KUKA KRL program: MyProgram_298().src

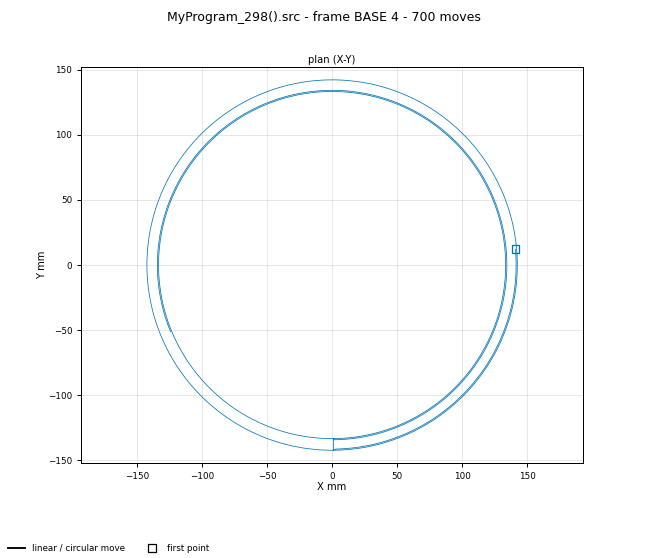
[picture p0: tool path of MyProgram_298().src in frame BASE 4, 700 of 700 moves have a stored position in this frame; points joined in program order, loops and branches not executed]
&ACCESS RVP
&REL 1
&PARAM TEMPLATE = C:\KRC\Roboter\Template\vorgabe
&PARAM EDITMASK = *
DEF MyProgram_298()
; ---- Setting reference (Base) ----
$BASE = BASE_DATA[4]

; --------------------------
; ---- Setting tool (TCP) ----
$TOOL = TOOL_DATA[3]
; --------------------------

$VEL.CP = VEL_APROX_PRINT
Startdeposition()
$VEL.CP = VEL_PRINT
LIN {X 140.7896,Y 12.0688,Z 178,A 6.9353,B 5.8277,C 0.252,E1 5.9925,E2 445.646} C_DIS
LIN {X 141.111,Y 7.4247,Z 178,A 5.2439,B 5.8277,C 0.2542,E1 5.9928,E2 447.3133} C_DIS
LIN {X 141.2495,Y 3.9929,Z 178,A 3.8231,B 5.8274,C 0.2586,E1 5.9929,E2 448.7388} C_DIS
LIN {X 141.3032,Y 0.9542,Z 178,A 2.4803,B 5.8272,C 0.2639,E1 5.9929,E2 450.0971} C_DIS
LIN {X 141.2517,Y -3.912,Z 178,A 0.8337,B 5.8272,C 0.2642,E1 5.9929,E2 451.7025} C_DIS
LIN {X 141.1557,Y -6.5363,Z 178,A -0.2484,B 5.827,C 0.2675,E1 5.9928,E2 452.7877} C_DIS
LIN {X 140.9501,Y -10.0235,Z 178,A -1.7448,B 5.8268,C 0.2729,E1 5.9925,E2 454.2957} C_DIS
LIN {X 140.6912,Y -13.1685,Z 178,A -2.8653,B 5.8268,C 0.2739,E1 5.9922,E2 455.3963} C_DIS
LIN {X 140.4174,Y -15.8362,Z 178,A -4.0893,B 5.8265,C 0.2793,E1 5.9919,E2 456.6392} C_DIS
LIN {X 139.8782,Y -20.0345,Z 178,A -5.6337,B 5.8264,C 0.2813,E1 5.9913,E2 458.1625} C_DIS
LIN {X 139.4162,Y -23.0315,Z 178,A -6.8756,B 5.8262,C 0.285,E1 5.9907,E2 459.407} C_DIS
LIN {X 138.9631,Y -25.6338,Z 178,A -7.9325,B 5.8261,C 0.2878,E1 5.9902,E2 460.4631} C_DIS
LIN {X 138.2972,Y -29.0141,Z 178,A -9.3188,B 5.8259,C 0.2915,E1 5.9895,E2 461.8492} C_DIS
LIN {X 137.5734,Y -32.2709,Z 178,A -10.7608,B 5.8256,C 0.2968,E1 5.9885,E2 463.3041} C_DIS
LIN {X 136.5863,Y -36.2143,Z 178,A -12.0709,B 5.8256,C 0.2958,E1 5.9877,E2 464.571} C_DIS
LIN {X 134.7,Y -42.6994,Z 178,A -14.9784,B 5.8251,C 0.3062,E1 5.9854,E2 467.5033} C_DIS
LIN {X 133.7418,Y -45.6164,Z 178,A -16.2242,B 5.825,C 0.3096,E1 5.9842,E2 468.7504} C_DIS
LIN {X 132.4239,Y -49.3072,Z 178,A -17.5833,B 5.825,C 0.3101,E1 5.983,E2 470.0805} C_DIS
LIN {X 131.439,Y -51.8799,Z 178,A -18.785,B 5.8247,C 0.3145,E1 5.9817,E2 471.2945} C_DIS
LIN {X 130.3827,Y -54.4752,Z 178,A -19.833,B 5.8247,C 0.3161,E1 5.9806,E2 472.3318} C_DIS
LIN {X 129.269,Y -57.0718,Z 178,A -21.1045,B 5.8243,C 0.3212,E1 5.9792,E2 473.621} C_DIS
LIN {X 127.8364,Y -60.2132,Z 178,A -22.518,B 5.8241,C 0.3251,E1 5.9775,E2 475.0377} C_DIS
LIN {X 126.2018,Y -63.5662,Z 178,A -23.9585,B 5.824,C 0.3278,E1 5.9758,E2 476.47} C_DIS
LIN {X 124.2714,Y -67.2649,Z 178,A -25.6148,B 5.8237,C 0.3316,E1 5.9736,E2 478.1232} C_DIS
LIN {X 122.0886,Y -71.1498,Z 178,A -27.2593,B 5.8237,C 0.3335,E1 5.9713,E2 479.7478} C_DIS
LIN {X 119.3608,Y -75.636,Z 178,A -29.4838,B 5.8232,C 0.3403,E1 5.9681,E2 481.987} C_DIS
LIN {X 116.8514,Y -79.4582,Z 178,A -31.2611,B 5.8231,C 0.3436,E1 5.9653,E2 483.7558} C_DIS
LIN {X 114.4302,Y -82.9065,Z 178,A -33.3278,B 5.8225,C 0.3534,E1 5.9619,E2 485.8715} C_DIS
LIN {X 111.8215,Y -86.3927,Z 178,A -34.7631,B 5.8225,C 0.3522,E1 5.9595,E2 487.2647} C_DIS
LIN {X 108.8999,Y -90.0476,Z 178,A -36.5124,B 5.8225,C 0.3542,E1 5.9564,E2 488.996} C_DIS
LIN {X 106.2988,Y -93.1042,Z 178,A -38.1229,B 5.8222,C 0.3575,E1 5.9535,E2 490.6058} C_DIS
LIN {X 103.2393,Y -96.4855,Z 178,A -39.9595,B 5.822,C 0.3613,E1 5.95,E2 492.4424} C_DIS
LIN {X 99.9844,Y -99.855,Z 178,A -41.8636,B 5.8217,C 0.3654,E1 5.9463,E2 494.3488} C_DIS
LIN {X 96.8119,Y -102.9333,Z 178,A -43.5703,B 5.8216,C 0.3677,E1 5.9429,E2 496.0457} C_DIS
LIN {X 93.3892,Y -106.0485,Z 178,A -45.543,B 5.8213,C 0.3729,E1 5.9387,E2 498.0328} C_DIS
LIN {X 89.623,Y -109.2499,Z 178,A -47.3778,B 5.8212,C 0.3741,E1 5.9349,E2 499.8468} C_DIS
LIN {X 86.4476,Y -111.7792,Z 178,A -48.9811,B 5.821,C 0.3765,E1 5.9313,E2 501.4458} C_DIS
LIN {X 82.9595,Y -114.3918,Z 178,A -50.6703,B 5.8209,C 0.3785,E1 5.9276,E2 503.1261} C_DIS
LIN {X 79.2176,Y -117.0142,Z 178,A -52.5363,B 5.8207,C 0.3818,E1 5.9233,E2 504.9954} C_DIS
LIN {X 75.9408,Y -119.1673,Z 178,A -54.1352,B 5.8205,C 0.3846,E1 5.9195,E2 506.5969} C_DIS
LIN {X 72.1514,Y -121.4989,Z 178,A -55.6674,B 5.8205,C 0.3833,E1 5.916,E2 508.0941} C_DIS
LIN {X 67.5081,Y -124.1388,Z 178,A -58.0661,B 5.8201,C 0.3901,E1 5.91,E2 510.5258} C_DIS
LIN {X 64.3589,Y -125.7982,Z 178,A -59.4105,B 5.8201,C 0.3906,E1 5.9067,E2 511.858} C_DIS
LIN {X 61.486,Y -127.2284,Z 178,A -60.7675,B 5.8199,C 0.3932,E1 5.9033,E2 513.2236} C_DIS
LIN {X 58.1815,Y -128.7726,Z 178,A -62.134,B 5.8199,C 0.3935,E1 5.8999,E2 514.5761} C_DIS
LIN {X 55.3271,Y -130.0261,Z 178,A -63.5794,B 5.8196,C 0.3977,E1 5.8961,E2 516.0468} C_DIS
LIN {X 51.3253,Y -131.6546,Z 178,A -65.0411,B 5.8198,C 0.3955,E1 5.8924,E2 517.4709} C_DIS
LIN {X 48.6469,Y -132.6698,Z 178,A -66.427,B 5.8195,C 0.4001,E1 5.8887,E2 518.8878} C_DIS
LIN {X 44.7714,Y -134.0252,Z 178,A -67.947,B 5.8195,C 0.3997,E1 5.8847,E2 520.3894} C_DIS
LIN {X 41.9416,Y -134.9389,Z 178,A -69.4697,B 5.8191,C 0.4055,E1 5.8806,E2 521.9554} C_DIS
LIN {X 38.5301,Y -135.9519,Z 178,A -70.6263,B 5.8193,C 0.4026,E1 5.8775,E2 523.0747} C_DIS
LIN {X 35.2419,Y -136.8412,Z 178,A -72.4658,B 5.8187,C 0.4104,E1 5.8724,E2 524.9762} C_DIS
LIN {X 30.6075,Y -137.9532,Z 178,A -74.0137,B 5.819,C 0.4063,E1 5.8683,E2 526.4742} C_DIS
LIN {X 27.1022,Y -138.6834,Z 178,A -75.2034,B 5.8192,C 0.4036,E1 5.8652,E2 527.6297} C_DIS
LIN {X 23.5539,Y -139.3291,Z 178,A -76.6385,B 5.8192,C 0.4041,E1 5.8612,E2 529.062} C_DIS
LIN {X 20.7157,Y -139.7809,Z 178,A -78.0954,B 5.8188,C 0.4089,E1 5.8571,E2 530.5587} C_DIS
LIN {X 16.6458,Y -140.3219,Z 178,A -79.5217,B 5.819,C 0.4063,E1 5.8532,E2 531.954} C_DIS
LIN {X 13.9017,Y -140.6208,Z 178,A -80.6337,B 5.819,C 0.4067,E1 5.8501,E2 533.0656} C_DIS
LIN {X 10.5102,Y -140.9146,Z 178,A -81.843,B 5.8191,C 0.4048,E1 5.8468,E2 534.2527} C_DIS
LIN {X 7.3431,Y -141.1151,Z 178,A -83.4444,B 5.8188,C 0.4095,E1 5.8422,E2 535.897} C_DIS
LIN {X 2.7408,Y -141.2798,Z 178,A -85.1904,B 5.8188,C 0.4082,E1 5.8374,E2 537.6277} C_DIS
LIN {X 2.7408,Y -141.2798,Z 178,A -85.1904,B 5.8188,C 0.4082,E1 5.8374,E2 537.6277} C_DIS
Enddeposition()
LIN {X 1.0318,Y -142.2048,Z 178,A -85.5763,B 5.819,C 0.4074,E1 5.8364,E2 538.0052} C_DIS
Startdeposition()
$VEL.CP = VEL_PRINT
LIN {X 3.8018,Y -142.1593,Z 178,A -84.2114,B 5.8193,C 0.4038,E1 5.8403,E2 536.606} C_DIS
LIN {X 7.0997,Y -142.0327,Z 178,A -82.8414,B 5.8193,C 0.4029,E1 5.8442,E2 535.2298} C_DIS
LIN {X 10.5794,Y -141.8161,Z 178,A -81.4286,B 5.8193,C 0.4023,E1 5.8481,E2 533.8152} C_DIS
LIN {X 13.9421,Y -141.5253,Z 178,A -80.075,B 5.8194,C 0.4019,E1 5.8519,E2 532.4617} C_DIS
LIN {X 17.7286,Y -141.1026,Z 178,A -78.5776,B 5.8194,C 0.4017,E1 5.856,E2 530.9687} C_DIS
LIN {X 20.9908,Y -140.6543,Z 178,A -77.2417,B 5.8194,C 0.4009,E1 5.8597,E2 529.6307} C_DIS
LIN {X 24.3237,Y -140.1162,Z 178,A -75.8217,B 5.8196,C 0.3992,E1 5.8636,E2 528.2017} C_DIS
LIN {X 27.858,Y -139.4554,Z 178,A -74.418,B 5.8196,C 0.3989,E1 5.8675,E2 526.8033} C_DIS
LIN {X 31.2944,Y -138.7243,Z 178,A -73.0141,B 5.8196,C 0.398,E1 5.8713,E2 525.4001} C_DIS
LIN {X 34.5683,Y -137.945,Z 178,A -71.6294,B 5.8198,C 0.3965,E1 5.8751,E2 524.0105} C_DIS
LIN {X 37.9249,Y -137.0601,Z 178,A -70.2819,B 5.8198,C 0.3961,E1 5.8787,E2 522.6691} C_DIS
LIN {X 41.789,Y -135.9313,Z 178,A -68.5849,B 5.82,C 0.3934,E1 5.8833,E2 520.9607} C_DIS
LIN {X 46.3797,Y -134.4342,Z 178,A -66.7442,B 5.82,C 0.393,E1 5.8881,E2 519.133} C_DIS
LIN {X 49.5577,Y -133.2956,Z 178,A -65.3978,B 5.82,C 0.3918,E1 5.8916,E2 517.7874} C_DIS
LIN {X 52.8099,Y -132.041,Z 178,A -64.0082,B 5.8202,C 0.3904,E1 5.8953,E2 516.3989} C_DIS
LIN {X 56.0719,Y -130.6892,Z 178,A -62.5985,B 5.8202,C 0.3888,E1 5.8989,E2 514.9898} C_DIS
LIN {X 59.2173,Y -129.2947,Z 178,A -61.2162,B 5.8204,C 0.3871,E1 5.9024,E2 513.607} C_DIS
LIN {X 62.3694,Y -127.8044,Z 178,A -59.845,B 5.8204,C 0.3857,E1 5.9058,E2 512.2393} C_DIS
LIN {X 65.496,Y -126.2311,Z 178,A -58.3602,B 5.8207,C 0.3826,E1 5.9096,E2 510.7433} C_DIS
LIN {X 69.4042,Y -124.1261,Z 178,A -56.6109,B 5.8208,C 0.3806,E1 5.9138,E2 508.998} C_DIS
LIN {X 73.1252,Y -121.9711,Z 178,A -54.9593,B 5.8209,C 0.3792,E1 5.9178,E2 507.356} C_DIS
LIN {X 76.0902,Y -120.1435,Z 178,A -53.5759,B 5.821,C 0.3772,E1 5.9211,E2 505.9741} C_DIS
LIN {X 79.0543,Y -118.214,Z 178,A -52.0494,B 5.8213,C 0.3732,E1 5.9246,E2 504.4326} C_DIS
LIN {X 82.6534,Y -115.7261,Z 178,A -50.4466,B 5.8213,C 0.3727,E1 5.9283,E2 502.8502} C_DIS
LIN {X 85.4653,Y -113.6656,Z 178,A -49.0809,B 5.8215,C 0.3708,E1 5.9313,E2 501.4885} C_DIS
LIN {X 88.6759,Y -111.1788,Z 178,A -47.4079,B 5.8217,C 0.3672,E1 5.935,E2 499.809} C_DIS
LIN {X 92.181,Y -108.2903,Z 178,A -45.6378,B 5.8218,C 0.3647,E1 5.9388,E2 498.0455} C_DIS
LIN {X 94.862,Y -105.9496,Z 178,A -44.2317,B 5.822,C 0.3623,E1 5.9417,E2 496.642} C_DIS
LIN {X 97.4308,Y -103.5925,Z 178,A -42.8526,B 5.8221,C 0.3598,E1 5.9445,E2 495.265} C_DIS
LIN {X 100.5199,Y -100.5984,Z 178,A -41.1447,B 5.8223,C 0.3567,E1 5.9479,E2 493.5591} C_DIS
LIN {X 103.0441,Y -98.0109,Z 178,A -39.729,B 5.8225,C 0.3542,E1 5.9507,E2 492.1476} C_DIS
LIN {X 105.4161,Y -95.4546,Z 178,A -38.3467,B 5.8227,C 0.3515,E1 5.9533,E2 490.7671} C_DIS
LIN {X 108.2186,Y -92.2654,Z 178,A -36.6624,B 5.8229,C 0.3482,E1 5.9564,E2 489.0848} C_DIS
LIN {X 110.5175,Y -89.499,Z 178,A -35.2473,B 5.823,C 0.3454,E1 5.9589,E2 487.673} C_DIS
LIN {X 112.6968,Y -86.7395,Z 178,A -33.7189,B 5.8233,C 0.3403,E1 5.9615,E2 486.1283} C_DIS
LIN {X 115.2677,Y -83.2918,Z 178,A -32.1596,B 5.8233,C 0.3391,E1 5.964,E2 484.5909} C_DIS
LIN {X 117.568,Y -80.0126,Z 178,A -30.4755,B 5.8237,C 0.3341,E1 5.9667,E2 482.8958} C_DIS
LIN {X 120.1428,Y -76.0912,Z 178,A -28.722,B 5.8238,C 0.3317,E1 5.9694,E2 481.159} C_DIS
LIN {X 122.116,Y -72.8822,Z 178,A -27.153,B 5.8241,C 0.327,E1 5.9716,E2 479.5816} C_DIS
LIN {X 124.1647,Y -69.3355,Z 178,A -25.5171,B 5.8243,C 0.3231,E1 5.9739,E2 477.9462} C_DIS
LIN {X 126.2634,Y -65.4346,Z 178,A -23.8758,B 5.8244,C 0.3209,E1 5.976,E2 476.3226} C_DIS
LIN {X 127.8295,Y -62.3186,Z 178,A -22.5037,B 5.8246,C 0.3178,E1 5.9777,E2 474.9537} C_DIS
LIN {X 129.3183,Y -59.1663,Z 178,A -21.1285,B 5.8248,C 0.3146,E1 5.9793,E2 473.5811} C_DIS
LIN {X 130.7514,Y -55.9279,Z 178,A -19.7382,B 5.8249,C 0.3114,E1 5.9809,E2 472.1945} C_DIS
LIN {X 132.0827,Y -52.7065,Z 178,A -18.3668,B 5.8251,C 0.3082,E1 5.9823,E2 470.8262} C_DIS
LIN {X 133.2951,Y -49.559,Z 178,A -17.0401,B 5.8253,C 0.3051,E1 5.9836,E2 469.5027} C_DIS
LIN {X 134.5104,Y -46.1599,Z 178,A -15.4987,B 5.8255,C 0.2997,E1 5.985,E2 467.9482} C_DIS
LIN {X 135.5815,Y -42.9116,Z 178,A -14.2649,B 5.8256,C 0.2983,E1 5.9861,E2 466.7327} C_DIS
LIN {X 136.6219,Y -39.4755,Z 178,A -12.8713,B 5.8258,C 0.2952,E1 5.9872,E2 465.3449} C_DIS
LIN {X 137.5474,Y -36.1194,Z 178,A -11.5022,B 5.8259,C 0.2919,E1 5.9882,E2 463.9791} C_DIS
LIN {X 138.3645,Y -32.8501,Z 178,A -10.1385,B 5.8261,C 0.288,E1 5.9891,E2 462.6133} C_DIS
LIN {X 139.1267,Y -29.4571,Z 178,A -8.8032,B 5.8263,C 0.2851,E1 5.9898,E2 461.2857} C_DIS
LIN {X 139.8334,Y -25.9021,Z 178,A -7.3729,B 5.8264,C 0.2815,E1 5.9906,E2 459.8581} C_DIS
LIN {X 140.4073,Y -22.5855,Z 178,A -6.0384,B 5.8266,C 0.2781,E1 5.9912,E2 458.5254} C_DIS
LIN {X 140.9181,Y -19.1361,Z 178,A -4.6369,B 5.8268,C 0.2741,E1 5.9918,E2 457.1232} C_DIS
LIN {X 141.356,Y -15.5658,Z 178,A -3.283,B 5.8269,C 0.2716,E1 5.9922,E2 455.7808} C_DIS
LIN {X 141.7303,Y -11.675,Z 178,A -1.7851,B 5.8271,C 0.2684,E1 5.9926,E2 454.2919} C_DIS
LIN {X 141.943,Y -8.7115,Z 178,A -0.5464,B 5.8272,C 0.2643,E1 5.9928,E2 453.0466} C_DIS
LIN {X 142.1185,Y -5.1195,Z 178,A 0.8518,B 5.8274,C 0.261,E1 5.993,E2 451.654} C_DIS
LIN {X 142.2072,Y -0.9928,Z 178,A 2.268,B 5.8274,C 0.2604,E1 5.993,E2 450.2694} C_DIS
LIN {X 142.199,Y 1.8524,Z 178,A 3.5882,B 5.8277,C 0.2542,E1 5.993,E2 448.9252} C_DIS
LIN {X 142.1137,Y 5.2435,Z 178,A 4.9594,B 5.8279,C 0.2502,E1 5.9929,E2 447.5523} C_DIS
LIN {X 141.8893,Y 9.577,Z 178,A 6.8418,B 5.8282,C 0.243,E1 5.9926,E2 445.6507} C_DIS
LIN {X 141.5259,Y 13.9363,Z 178,A 8.3626,B 5.8282,C 0.242,E1 5.9922,E2 444.1608} C_DIS
LIN {X 141.1269,Y 17.531,Z 178,A 9.7666,B 5.8283,C 0.2388,E1 5.9917,E2 442.7628} C_DIS
LIN {X 140.6554,Y 20.984,Z 178,A 11.1263,B 5.8285,C 0.2355,E1 5.9912,E2 441.4081} C_DIS
LIN {X 140.1177,Y 24.3154,Z 178,A 12.5193,B 5.8286,C 0.2312,E1 5.9905,E2 440.0097} C_DIS
LIN {X 139.4419,Y 27.9246,Z 178,A 13.9069,B 5.8288,C 0.2285,E1 5.9898,E2 438.6332} C_DIS
LIN {X 138.7328,Y 31.2573,Z 178,A 15.2662,B 5.8288,C 0.2249,E1 5.989,E2 437.2747} C_DIS
LIN {X 137.9528,Y 34.5376,Z 178,A 16.62,B 5.829,C 0.2213,E1 5.9881,E2 435.9207} C_DIS
LIN {X 136.8515,Y 38.6708,Z 178,A 18.1868,B 5.8291,C 0.2191,E1 5.987,E2 434.3735} C_DIS
LIN {X 136.0528,Y 41.392,Z 178,A 19.3635,B 5.8293,C 0.2154,E1 5.986,E2 433.1915} C_DIS
LIN {X 135.032,Y 44.6102,Z 178,A 20.7434,B 5.8293,C 0.2114,E1 5.9848,E2 431.8083} C_DIS
LIN {X 133.8596,Y 48.013,Z 178,A 22.1484,B 5.8295,C 0.2083,E1 5.9835,E2 430.4084} C_DIS
LIN {X 132.6757,Y 51.1942,Z 178,A 23.47,B 5.8296,C 0.2054,E1 5.9822,E2 429.0921} C_DIS
LIN {X 131.3819,Y 54.4291,Z 178,A 24.8413,B 5.8297,C 0.2022,E1 5.9808,E2 427.7242} C_DIS
LIN {X 129.9867,Y 57.6818,Z 178,A 26.3148,B 5.8299,C 0.1977,E1 5.9791,E2 426.2437} C_DIS
LIN {X 128.5349,Y 60.8488,Z 178,A 27.5899,B 5.8299,C 0.1962,E1 5.9776,E2 424.9848} C_DIS
LIN {X 127.0309,Y 63.9307,Z 178,A 28.9598,B 5.83,C 0.1928,E1 5.9759,E2 423.6159} C_DIS
LIN {X 125.3934,Y 67.0872,Z 178,A 30.4698,B 5.8302,C 0.188,E1 5.9739,E2 422.095} C_DIS
LIN {X 123.3001,Y 70.8619,Z 178,A 32.0718,B 5.8302,C 0.1859,E1 5.9718,E2 420.5102} C_DIS
LIN {X 121.5257,Y 73.863,Z 178,A 33.4534,B 5.8304,C 0.1828,E1 5.9698,E2 419.131} C_DIS
LIN {X 119.2361,Y 77.504,Z 178,A 35.159,B 5.8304,C 0.1791,E1 5.9672,E2 417.4282} C_DIS
LIN {X 116.8061,Y 81.1201,Z 178,A 36.8825,B 5.8306,C 0.1754,E1 5.9645,E2 415.7083} C_DIS
LIN {X 114.7097,Y 84.0585,Z 178,A 38.3768,B 5.8307,C 0.1714,E1 5.9621,E2 414.2082} C_DIS
LIN {X 112.0833,Y 87.5306,Z 178,A 40.0033,B 5.8307,C 0.1695,E1 5.9593,E2 412.5978} C_DIS
LIN {X 109.8763,Y 90.2855,Z 178,A 41.5412,B 5.8309,C 0.1645,E1 5.9566,E2 411.0444} C_DIS
LIN {X 107.042,Y 93.6278,Z 178,A 43.2608,B 5.8309,C 0.1614,E1 5.9534,E2 409.3302} C_DIS
LIN {X 104.1886,Y 96.793,Z 178,A 44.8289,B 5.831,C 0.1601,E1 5.9505,E2 407.7811} C_DIS
LIN {X 101.7452,Y 99.3586,Z 178,A 46.2987,B 5.8311,C 0.1565,E1 5.9477,E2 406.3055} C_DIS
LIN {X 98.6592,Y 102.4237,Z 178,A 47.9572,B 5.8311,C 0.1545,E1 5.9444,E2 404.6588} C_DIS
LIN {X 95.5257,Y 105.3516,Z 178,A 49.6621,B 5.8313,C 0.1514,E1 5.9409,E2 402.9565} C_DIS
LIN {X 91.9966,Y 108.4471,Z 178,A 51.602,B 5.8313,C 0.1472,E1 5.9368,E2 401.01} C_DIS
LIN {X 88.8163,Y 111.067,Z 178,A 53.1334,B 5.8313,C 0.1461,E1 5.9335,E2 399.4951} C_DIS
LIN {X 86.1098,Y 113.1784,Z 178,A 54.5078,B 5.8314,C 0.1438,E1 5.9304,E2 398.1216} C_DIS
LIN {X 83.3077,Y 115.2561,Z 178,A 56.015,B 5.8315,C 0.1399,E1 5.927,E2 396.6011} C_DIS
LIN {X 79.7275,Y 117.761,Z 178,A 57.622,B 5.8315,C 0.1393,E1 5.9234,E2 395.0139} C_DIS
LIN {X 76.7708,Y 119.7096,Z 178,A 59.0155,B 5.8315,C 0.1376,E1 5.9201,E2 393.6246} C_DIS
LIN {X 73.8139,Y 121.5554,Z 178,A 60.4867,B 5.8317,C 0.1345,E1 5.9166,E2 392.1448} C_DIS
LIN {X 70.0937,Y 123.7384,Z 178,A 62.2577,B 5.8317,C 0.1315,E1 5.9123,E2 390.3695} C_DIS
LIN {X 66.2699,Y 125.8248,Z 178,A 63.8719,B 5.8317,C 0.1311,E1 5.9084,E2 388.7734} C_DIS
LIN {X 63.0883,Y 127.4498,Z 178,A 65.2721,B 5.8317,C 0.1298,E1 5.9049,E2 387.3783} C_DIS
LIN {X 59.9571,Y 128.9527,Z 178,A 66.6575,B 5.8318,C 0.1283,E1 5.9014,E2 385.9949} C_DIS
LIN {X 57.5272,Y 130.0558,Z 178,A 67.7427,B 5.8318,C 0.1269,E1 5.8986,E2 384.9085} C_DIS
LIN {X 53.9852,Y 131.5672,Z 178,A 69.2765,B 5.8318,C 0.1254,E1 5.8947,E2 383.3772} C_DIS
LIN {X 51.072,Y 132.7233,Z 178,A 70.5185,B 5.8318,C 0.1243,E1 5.8914,E2 382.138} C_DIS
LIN {X 47.2351,Y 134.1376,Z 178,A 72.2781,B 5.832,C 0.1211,E1 5.8868,E2 380.3642} C_DIS
LIN {X 43.3592,Y 135.4385,Z 178,A 73.8744,B 5.832,C 0.1203,E1 5.8826,E2 378.7748} C_DIS
LIN {X 39.5047,Y 136.6133,Z 178,A 75.4664,B 5.832,C 0.1194,E1 5.8783,E2 377.1871} C_DIS
LIN {X 36.119,Y 137.5475,Z 178,A 76.8008,B 5.832,C 0.1194,E1 5.8747,E2 375.8635} C_DIS
LIN {X 32.8433,Y 138.3661,Z 178,A 78.159,B 5.832,C 0.1185,E1 5.871,E2 374.5059} C_DIS
LIN {X 29.4441,Y 139.1295,Z 178,A 79.5529,B 5.832,C 0.1178,E1 5.8672,E2 373.1137} C_DIS
LIN {X 25.9185,Y 139.8303,Z 178,A 80.9981,B 5.832,C 0.117,E1 5.8633,E2 371.6693} C_DIS
LIN {X 22.2652,Y 140.457,Z 178,A 82.3946,B 5.832,C 0.1176,E1 5.8595,E2 370.2857} C_DIS
LIN {X 19.1288,Y 140.9191,Z 178,A 83.8019,B 5.832,C 0.1153,E1 5.8555,E2 368.8621} C_DIS
LIN {X 15.557,Y 141.3569,Z 178,A 85.1854,B 5.832,C 0.1156,E1 5.8517,E2 367.4876} C_DIS
LIN {X 12.1982,Y 141.6861,Z 178,A 86.5867,B 5.832,C 0.1147,E1 5.8478,E2 366.0814} C_DIS
LIN {X 8.7224,Y 141.9423,Z 178,A 87.9783,B 5.832,C 0.1145,E1 5.8439,E2 364.692} C_DIS
LIN {X 5.1123,Y 142.1188,Z 178,A 89.3938,B 5.832,C 0.1149,E1 5.84,E2 363.2824} C_DIS
LIN {X 1.6282,Y 142.2027,Z 178,A 90.795,B 5.832,C 0.1148,E1 5.8361,E2 361.8822} C_DIS
LIN {X -1.8595,Y 142.1989,Z 178,A 92.2118,B 5.832,C 0.1146,E1 5.8321,E2 360.4646} C_DIS
LIN {X -5.2331,Y 142.1141,Z 178,A 93.6179,B 5.8321,C 0.1141,E1 5.8282,E2 359.053} C_DIS
LIN {X -8.7251,Y 141.9421,Z 178,A 95.014,B 5.8321,C 0.1144,E1 5.8243,E2 357.6592} C_DIS
LIN {X -12.3225,Y 141.6756,Z 178,A 96.4505,B 5.8321,C 0.1149,E1 5.8203,E2 356.2256} C_DIS
LIN {X -15.6804,Y 141.3436,Z 178,A 97.812,B 5.8321,C 0.1153,E1 5.8165,E2 354.8646} C_DIS
LIN {X -19.2495,Y 140.9032,Z 178,A 99.2796,B 5.8321,C 0.1155,E1 5.8125,E2 353.3954} C_DIS
LIN {X -22.6275,Y 140.4004,Z 178,A 100.6613,B 5.8321,C 0.116,E1 5.8086,E2 352.0137} C_DIS
LIN {X -26.1702,Y 139.7821,Z 178,A 102.11,B 5.8321,C 0.1167,E1 5.8047,E2 350.5659} C_DIS
LIN {X -29.5798,Y 139.1002,Z 178,A 103.5149,B 5.8321,C 0.1174,E1 5.8008,E2 349.1613} C_DIS
LIN {X -32.9661,Y 138.3365,Z 178,A 104.8898,B 5.8321,C 0.1186,E1 5.7971,E2 347.7902} C_DIS
LIN {X -36.3319,Y 137.4907,Z 178,A 106.3064,B 5.832,C 0.1193,E1 5.7933,E2 346.3721} C_DIS
LIN {X -39.9883,Y 136.4717,Z 178,A 107.8081,B 5.832,C 0.1208,E1 5.7892,E2 344.8749} C_DIS
LIN {X -42.95,Y 135.5692,Z 178,A 109.1216,B 5.832,C 0.121,E1 5.7857,E2 343.5538} C_DIS
LIN {X -46.3741,Y 134.4361,Z 178,A 110.5892,B 5.832,C 0.1221,E1 5.7818,E2 342.0852} C_DIS
LIN {X -49.5676,Y 133.2919,Z 178,A 112.0314,B 5.832,C 0.1225,E1 5.778,E2 340.6343} C_DIS
LIN {X -52.8178,Y 132.0378,Z 178,A 113.3778,B 5.8319,C 0.1247,E1 5.7745,E2 339.2962} C_DIS
LIN {X -56.0356,Y 130.7049,Z 178,A 114.8084,B 5.8319,C 0.1259,E1 5.7709,E2 337.8631} C_DIS
LIN {X -59.2195,Y 129.2937,Z 178,A 116.2254,B 5.8319,C 0.1273,E1 5.7672,E2 336.4454} C_DIS
LIN {X -62.3688,Y 127.8047,Z 178,A 117.6316,B 5.8318,C 0.129,E1 5.7637,E2 335.0398} C_DIS
LIN {X -65.4985,Y 126.2298,Z 178,A 119.0537,B 5.8318,C 0.1307,E1 5.7602,E2 333.6175} C_DIS
LIN {X -68.623,Y 124.5596,Z 178,A 120.4854,B 5.8318,C 0.1325,E1 5.7567,E2 332.1864} C_DIS
LIN {X -71.6092,Y 122.8675,Z 178,A 121.9101,B 5.8317,C 0.134,E1 5.7532,E2 330.7572} C_DIS
LIN {X -74.6483,Y 121.0449,Z 178,A 123.3484,B 5.8317,C 0.136,E1 5.7498,E2 329.3187} C_DIS
LIN {X -77.5943,Y 119.1775,Z 178,A 124.7777,B 5.8316,C 0.1378,E1 5.7464,E2 327.8874} C_DIS
LIN {X -80.629,Y 117.1457,Z 178,A 126.3956,B 5.8316,C 0.1385,E1 5.7426,E2 326.2518} C_DIS
LIN {X -84.0833,Y 114.6915,Z 178,A 127.9956,B 5.8315,C 0.1425,E1 5.739,E2 324.6671} C_DIS
LIN {X -86.8207,Y 112.634,Z 178,A 129.3938,B 5.8315,C 0.1447,E1 5.7359,E2 323.2676} C_DIS
LIN {X -89.5924,Y 110.4422,Z 178,A 130.8551,B 5.8314,C 0.1468,E1 5.7327,E2 321.8026} C_DIS
LIN {X -92.2978,Y 108.191,Z 178,A 132.4283,B 5.8314,C 0.1477,E1 5.7293,E2 320.2106} C_DIS
LIN {X -95.5623,Y 105.3184,Z 178,A 134.201,B 5.8313,C 0.1508,E1 5.7256,E2 318.4366} C_DIS
LIN {X -98.74,Y 102.3455,Z 178,A 135.9818,B 5.8312,C 0.1539,E1 5.722,E2 316.6538} C_DIS
LIN {X -101.7853,Y 99.3176,Z 178,A 137.632,B 5.8311,C 0.1583,E1 5.7188,E2 315.0155} C_DIS
LIN {X -104.2254,Y 96.7535,Z 178,A 139.0775,B 5.8311,C 0.161,E1 5.7161,E2 313.5687} C_DIS
LIN {X -106.5991,Y 94.1316,Z 178,A 140.6525,B 5.831,C 0.1624,E1 5.7131,E2 311.9755} C_DIS
LIN {X -109.3867,Y 90.8775,Z 178,A 142.2987,B 5.8308,C 0.167,E1 5.7102,E2 310.3412} C_DIS
LIN {X -111.6042,Y 88.1406,Z 178,A 143.7183,B 5.8308,C 0.1702,E1 5.7077,E2 308.9229} C_DIS
LIN {X -114.1733,Y 84.7857,Z 178,A 145.4784,B 5.8306,C 0.1735,E1 5.7047,E2 307.1568} C_DIS
LIN {X -116.2702,Y 81.8863,Z 178,A 146.9347,B 5.8306,C 0.1766,E1 5.7023,E2 305.6999} C_DIS
LIN {X -118.2437,Y 79.0098,Z 178,A 148.3807,B 5.8305,C 0.1795,E1 5.7001,E2 304.2498} C_DIS
LIN {X -120.1518,Y 76.0769,Z 178,A 149.818,B 5.8304,C 0.1826,E1 5.6979,E2 302.8103} C_DIS
LIN {X -122.0099,Y 73.0602,Z 178,A 151.2626,B 5.8303,C 0.1859,E1 5.6958,E2 301.3647} C_DIS
LIN {X -123.7376,Y 70.0951,Z 178,A 152.6857,B 5.8302,C 0.1889,E1 5.6938,E2 299.9376} C_DIS
LIN {X -125.4359,Y 67.008,Z 178,A 154.1502,B 5.8301,C 0.192,E1 5.6919,E2 298.4685} C_DIS
LIN {X -127.0653,Y 63.863,Z 178,A 155.5984,B 5.83,C 0.1955,E1 5.69,E2 297.0188} C_DIS
LIN {X -128.5902,Y 60.7331,Z 178,A 157.1545,B 5.8299,C 0.1975,E1 5.6881,E2 295.444} C_DIS
LIN {X -130.0582,Y 57.5219,Z 178,A 158.4855,B 5.8297,C 0.2021,E1 5.6866,E2 294.1262} C_DIS
LIN {X -131.4245,Y 54.327,Z 178,A 159.9187,B 5.8297,C 0.2055,E1 5.6851,E2 292.6899} C_DIS
LIN {X -132.7224,Y 51.0741,Z 178,A 161.3508,B 5.8295,C 0.209,E1 5.6836,E2 291.2563} C_DIS
LIN {X -133.8959,Y 47.9121,Z 178,A 162.7641,B 5.8294,C 0.2121,E1 5.6823,E2 289.837} C_DIS
LIN {X -135.0686,Y 44.5003,Z 178,A 164.229,B 5.8292,C 0.2159,E1 5.681,E2 288.372} C_DIS
LIN {X -136.1189,Y 41.176,Z 178,A 165.677,B 5.8292,C 0.2193,E1 5.6798,E2 286.9195} C_DIS
LIN {X -137.0573,Y 37.9346,Z 178,A 167.0802,B 5.829,C 0.2226,E1 5.6787,E2 285.5118} C_DIS
LIN {X -137.9463,Y 34.5632,Z 178,A 168.5089,B 5.8288,C 0.2263,E1 5.6777,E2 284.0812} C_DIS
LIN {X -138.8779,Y 30.6095,Z 178,A 170.0941,B 5.8286,C 0.2314,E1 5.6767,E2 282.5041} C_DIS
LIN {X -139.4861,Y 27.7076,Z 178,A 171.4085,B 5.8286,C 0.2335,E1 5.676,E2 281.1751} C_DIS
LIN {X -140.1411,Y 24.1817,Z 178,A 172.8685,B 5.8284,C 0.2374,E1 5.6753,E2 279.7144} C_DIS
LIN {X -140.6746,Y 20.8532,Z 178,A 174.2984,B 5.8283,C 0.2405,E1 5.6746,E2 278.2762} C_DIS
LIN {X -141.1546,Y 17.2988,Z 178,A 175.7859,B 5.8281,C 0.2442,E1 5.6741,E2 276.7843} C_DIS
LIN {X -141.5287,Y 13.9075,Z 178,A 177.1841,B 5.828,C 0.2478,E1 5.6737,E2 275.3841} C_DIS
LIN {X -141.8345,Y 10.328,Z 178,A 178.6416,B 5.8278,C 0.2518,E1 5.6734,E2 273.9265} C_DIS
LIN {X -142.045,Y 6.8548,Z 178,A -179.9112,B 5.8276,C 0.2554,E1 5.6732,E2 272.4745} C_DIS
LIN {X -142.168,Y 3.4889,Z 178,A -178.4178,B 5.8276,C 0.2579,E1 5.673,E2 270.9642} C_DIS
LIN {X -142.2123,Y -0.0237,Z 178,A -176.9975,B 5.8274,C 0.2618,E1 5.673,E2 269.5444} C_DIS
LIN {X -142.1674,Y -3.5132,Z 178,A -175.6025,B 5.8272,C 0.266,E1 5.6731,E2 268.152} C_DIS
LIN {X -142.0326,Y -7.102,Z 178,A -174.1506,B 5.827,C 0.27,E1 5.6733,E2 266.7005} C_DIS
LIN {X -141.8166,Y -10.5734,Z 178,A -172.691,B 5.8268,C 0.2734,E1 5.6736,E2 265.2342} C_DIS
LIN {X -141.5165,Y -14.0338,Z 178,A -171.2697,B 5.8267,C 0.2772,E1 5.6739,E2 263.811} C_DIS
LIN {X -141.1207,Y -17.5831,Z 178,A -169.7956,B 5.8265,C 0.2809,E1 5.6744,E2 262.3334} C_DIS
LIN {X -140.6498,Y -21.0198,Z 178,A -168.3818,B 5.8263,C 0.2846,E1 5.675,E2 260.9185} C_DIS
LIN {X -140.0696,Y -24.5843,Z 178,A -166.8986,B 5.8261,C 0.2884,E1 5.6757,E2 259.4325} C_DIS
LIN {X -139.456,Y -27.8551,Z 178,A -165.4784,B 5.826,C 0.2913,E1 5.6764,E2 258.0028} C_DIS
LIN {X -138.7306,Y -31.267,Z 178,A -164.0402,B 5.8258,C 0.2949,E1 5.6773,E2 256.5611} C_DIS
LIN {X -137.9493,Y -34.5516,Z 178,A -162.6164,B 5.8256,C 0.298,E1 5.6782,E2 255.1297} C_DIS
LIN {X -137.0568,Y -37.9364,Z 178,A -161.1406,B 5.8255,C 0.3012,E1 5.6793,E2 253.6461} C_DIS
LIN {X -136.053,Y -41.3912,Z 178,A -159.7478,B 5.8252,C 0.3057,E1 5.6804,E2 252.2618} C_DIS
LIN {X -135.0327,Y -44.6081,Z 178,A -158.2209,B 5.8252,C 0.3076,E1 5.6818,E2 250.7135} C_DIS
LIN {X -133.8454,Y -48.0524,Z 178,A -156.8532,B 5.8249,C 0.3126,E1 5.683,E2 249.36} C_DIS
LIN {X -132.6699,Y -51.2091,Z 178,A -155.4399,B 5.8247,C 0.3155,E1 5.6844,E2 247.94} C_DIS
LIN {X -131.3803,Y -54.4329,Z 178,A -154.0098,B 5.8245,C 0.3189,E1 5.6859,E2 246.5065} C_DIS
LIN {X -129.9904,Y -57.6735,Z 178,A -152.5673,B 5.8243,C 0.3223,E1 5.6876,E2 245.0619} C_DIS
LIN {X -128.5316,Y -60.8558,Z 178,A -151.131,B 5.8242,C 0.3256,E1 5.6893,E2 243.6229} C_DIS
LIN {X -127.0262,Y -63.9398,Z 178,A -149.7028,B 5.824,C 0.3286,E1 5.691,E2 242.1893} C_DIS
LIN {X -125.382,Y -67.1084,Z 178,A -148.229,B 5.8238,C 0.3318,E1 5.693,E2 240.7115} C_DIS
LIN {X -123.3258,Y -70.8169,Z 178,A -146.4691,B 5.8236,C 0.3354,E1 5.6954,E2 238.9454} C_DIS
LIN {X -121.5264,Y -73.8618,Z 178,A -145.0136,B 5.8234,C 0.3385,E1 5.6975,E2 237.4866} C_DIS
LIN {X -119.233,Y -77.5088,Z 178,A -143.2325,B 5.8232,C 0.3421,E1 5.7002,E2 235.7} C_DIS
LIN {X -116.8013,Y -81.1271,Z 178,A -141.4387,B 5.823,C 0.3458,E1 5.703,E2 233.902} C_DIS
LIN {X -114.7109,Y -84.0569,Z 178,A -139.9842,B 5.8228,C 0.349,E1 5.7054,E2 232.4474} C_DIS
LIN {X -112.6493,Y -86.801,Z 178,A -138.5721,B 5.8226,C 0.3517,E1 5.7078,E2 231.0319} C_DIS
LIN {X -110.4513,Y -89.5811,Z 178,A -137.1143,B 5.8225,C 0.3545,E1 5.7103,E2 229.5705} C_DIS
LIN {X -108.2098,Y -92.2756,Z 178,A -135.5352,B 5.8225,C 0.3556,E1 5.7132,E2 227.9694} C_DIS
LIN {X -105.331,Y -95.5484,Z 178,A -133.7561,B 5.8222,C 0.3589,E1 5.7165,E2 226.1876} C_DIS
LIN {X -102.223,Y -98.8665,Z 178,A -131.9257,B 5.822,C 0.3626,E1 5.72,E2 224.3579} C_DIS
LIN {X -99.3206,Y -101.7825,Z 178,A -130.3251,B 5.8217,C 0.3665,E1 5.7232,E2 222.7653} C_DIS
LIN {X -96.7954,Y -104.1864,Z 178,A -128.7959,B 5.8217,C 0.3676,E1 5.7264,E2 221.2196} C_DIS
LIN {X -93.5431,Y -107.1159,Z 178,A -127.1084,B 5.8214,C 0.3717,E1 5.7299,E2 219.5427} C_DIS
LIN {X -90.2592,Y -109.8978,Z 178,A -125.3356,B 5.8212,C 0.3743,E1 5.7337,E2 217.7649} C_DIS
LIN {X -87.3206,Y -112.2466,Z 178,A -123.7034,B 5.8212,C 0.3755,E1 5.7373,E2 216.1171} C_DIS
LIN {X -84.0043,Y -114.7495,Z 178,A -122.0178,B 5.821,C 0.378,E1 5.7411,E2 214.4302} C_DIS
LIN {X -80.4505,Y -117.2682,Z 178,A -120.3428,B 5.8208,C 0.3817,E1 5.7449,E2 212.7661} C_DIS
LIN {X -77.5069,Y -119.2343,Z 178,A -118.7672,B 5.8208,C 0.382,E1 5.7486,E2 211.1703} C_DIS
LIN {X -73.8081,Y -121.5589,Z 178,A -117.1197,B 5.8205,C 0.3858,E1 5.7525,E2 209.5381} C_DIS
LIN {X -70.5119,Y -123.4998,Z 178,A -115.4566,B 5.8205,C 0.3864,E1 5.7566,E2 207.8585} C_DIS
LIN {X -67.0387,Y -125.4194,Z 178,A -113.9181,B 5.8203,C 0.3891,E1 5.7603,E2 206.3281} C_DIS
LIN {X -63.8841,Y -127.0546,Z 178,A -112.4863,B 5.8202,C 0.3908,E1 5.7639,E2 204.8961} C_DIS
LIN {X -60.7515,Y -128.5814,Z 178,A -111.0704,B 5.8201,C 0.3923,E1 5.7674,E2 203.4785} C_DIS
LIN {X -57.0999,Y -130.2447,Z 178,A -109.497,B 5.8199,C 0.3945,E1 5.7714,E2 201.9108} C_DIS
LIN {X -54.3139,Y -131.43,Z 178,A -108.2106,B 5.8199,C 0.3949,E1 5.7748,E2 200.6152} C_DIS
LIN {X -50.8679,Y -132.8026,Z 178,A -106.7034,B 5.8198,C 0.3961,E1 5.7787,E2 199.1061} C_DIS
LIN {X -47.4507,Y -134.0623,Z 178,A -105.063,B 5.8198,C 0.3952,E1 5.7831,E2 197.442} C_DIS
LIN {X -43.1883,Y -135.4931,Z 178,A -103.3225,B 5.8198,C 0.3975,E1 5.7877,E2 195.7107} C_DIS
LIN {X -39.4847,Y -136.6192,Z 178,A -101.8459,B 5.8196,C 0.3996,E1 5.7916,E2 194.2451} C_DIS
LIN {X -36.1243,Y -137.5461,Z 178,A -100.4342,B 5.8196,C 0.4004,E1 5.7954,E2 192.8321} C_DIS
LIN {X -32.8497,Y -138.3646,Z 178,A -99.0613,B 5.8195,C 0.401,E1 5.7991,E2 191.457} C_DIS
LIN {X -29.4501,Y -139.1282,Z 178,A -97.6535,B 5.8195,C 0.4016,E1 5.803,E2 190.0483} C_DIS
LIN {X -25.9225,Y -139.8295,Z 178,A -96.1923,B 5.8194,C 0.4021,E1 5.807,E2 188.585} C_DIS
LIN {X -22.5839,Y -140.4076,Z 178,A -94.812,B 5.8194,C 0.4024,E1 5.8108,E2 187.2022} C_DIS
LIN {X -19.1331,Y -140.9185,Z 178,A -93.3726,B 5.8194,C 0.4023,E1 5.8148,E2 185.7576} C_DIS
LIN {X -15.5613,Y -141.3564,Z 178,A -91.9821,B 5.8194,C 0.4034,E1 5.8187,E2 184.3747} C_DIS
LIN {X -12.2023,Y -141.6857,Z 178,A -90.5715,B 5.8194,C 0.4029,E1 5.8226,E2 182.9566} C_DIS
LIN {X -8.7093,Y -141.9431,Z 178,A -89.1766,B 5.8194,C 0.4032,E1 5.8265,E2 181.5633} C_DIS
LIN {X -4.5869,Y -142.1375,Z 178,A -87.6089,B 5.8192,C 0.4045,E1 5.8308,E2 180.0079} C_DIS
LIN {X -1.6314,Y -142.2026,Z 178,A -86.3619,B 5.8192,C 0.4036,E1 5.8343,E2 178.7527} C_DIS
LIN {X 1.0318,Y -142.2048,Z 178,A -85.576,B 5.819,C 0.4075,E1 5.8364,E2 178.0051} C_DIS
Enddeposition()
LIN {X 0.9647,Y -133.2696,Z 179,A -85.7811,B 5.8301,C 0.3767,E1 5.8457,E2 177.904} C_DIS
Startdeposition()
$VEL.CP = VEL_PRINT
LIN {X -2.1693,Y -133.2586,Z 179,A -87.6034,B 5.8297,C 0.383,E1 5.8404,E2 179.7865} C_DIS
LIN {X -6.5493,Y -133.1152,Z 179,A -89.4902,B 5.8297,C 0.383,E1 5.8351,E2 181.6744} C_DIS
LIN {X -10.9307,Y -132.8274,Z 179,A -91.3073,B 5.8297,C 0.382,E1 5.8301,E2 183.4836} C_DIS
LIN {X -14.0283,Y -132.5359,Z 179,A -92.68,B 5.8297,C 0.3822,E1 5.8263,E2 184.8611} C_DIS
LIN {X -17.4444,Y -132.1295,Z 179,A -94.1198,B 5.8297,C 0.3814,E1 5.8223,E2 186.2967} C_DIS
LIN {X -21.179,Y -131.5847,Z 179,A -95.7297,B 5.8298,C 0.3807,E1 5.8179,E2 187.9056} C_DIS
LIN {X -24.3967,Y -131.0255,Z 179,A -97.1666,B 5.8298,C 0.3806,E1 5.8139,E2 189.3471} C_DIS
LIN {X -27.5991,Y -130.3881,Z 179,A -98.4606,B 5.83,C 0.3786,E1 5.8104,E2 190.6278} C_DIS
LIN {X -30.2894,Y -129.7899,Z 179,A -99.8791,B 5.8298,C 0.3808,E1 5.8064,E2 192.0757} C_DIS
LIN {X -33.7108,Y -128.9436,Z 179,A -101.3285,B 5.8299,C 0.3791,E1 5.8025,E2 193.5174} C_DIS
LIN {X -36.8628,Y -128.0779,Z 179,A -102.7922,B 5.8299,C 0.3789,E1 5.7986,E2 194.9887} C_DIS
LIN {X -40.7944,Y -126.8791,Z 179,A -104.5382,B 5.83,C 0.3774,E1 5.7939,E2 196.7323} C_DIS
LIN {X -44.4259,Y -125.656,Z 179,A -106.3765,B 5.83,C 0.3782,E1 5.789,E2 198.5947} C_DIS
LIN {X -49.0269,Y -123.9331,Z 179,A -108.2651,B 5.8303,C 0.3737,E1 5.7842,E2 200.4559} C_DIS
LIN {X -52.5139,Y -122.4943,Z 179,A -109.8941,B 5.8303,C 0.3722,E1 5.78,E2 202.086} C_DIS
LIN {X -55.5013,Y -121.1703,Z 179,A -111.3105,B 5.8305,C 0.3708,E1 5.7764,E2 203.504} C_DIS
LIN {X -58.4536,Y -119.7743,Z 179,A -112.7271,B 5.8305,C 0.3694,E1 5.7728,E2 204.9223} C_DIS
LIN {X -61.3715,Y -118.3062,Z 179,A -114.2383,B 5.8305,C 0.3689,E1 5.769,E2 206.4468} C_DIS
LIN {X -65.1142,Y -116.289,Z 179,A -116.1218,B 5.8307,C 0.3672,E1 5.7644,E2 208.3373} C_DIS
LIN {X -68.5257,Y -114.3122,Z 179,A -117.7204,B 5.8309,C 0.3639,E1 5.7605,E2 209.924} C_DIS
LIN {X -71.7363,Y -112.3248,Z 179,A -119.4668,B 5.8309,C 0.3629,E1 5.7564,E2 211.6855} C_DIS
LIN {X -74.9772,Y -110.1883,Z 179,A -121.1577,B 5.8311,C 0.3606,E1 5.7525,E2 213.3791} C_DIS
LIN {X -78.0685,Y -108.0198,Z 179,A -122.792,B 5.8312,C 0.3582,E1 5.7487,E2 215.0147} C_DIS
LIN {X -81.358,Y -105.5649,Z 179,A -124.6066,B 5.8314,C 0.3559,E1 5.7447,E2 216.8353} C_DIS
LIN {X -84.5518,Y -103.0242,Z 179,A -126.3067,B 5.8316,C 0.3523,E1 5.741,E2 218.5285} C_DIS
LIN {X -87.6721,Y -100.382,Z 179,A -128.1013,B 5.8318,C 0.3496,E1 5.7372,E2 220.3273} C_DIS
LIN {X -90.7185,Y -97.6377,Z 179,A -129.9476,B 5.8319,C 0.3472,E1 5.7334,E2 222.1835} C_DIS
LIN {X -93.8463,Y -94.6352,Z 179,A -131.8414,B 5.8321,C 0.3439,E1 5.7296,E2 224.0806} C_DIS
LIN {X -96.9114,Y -91.4938,Z 179,A -133.7098,B 5.8323,C 0.34,E1 5.726,E2 225.9463} C_DIS
LIN {X -99.6757,Y -88.4746,Z 179,A -135.5574,B 5.8325,C 0.3373,E1 5.7225,E2 227.8041} C_DIS
LIN {X -102.4868,Y -85.2024,Z 179,A -137.46,B 5.8327,C 0.3338,E1 5.719,E2 229.7122} C_DIS
LIN {X -105.2256,Y -81.7957,Z 179,A -139.3792,B 5.8329,C 0.3301,E1 5.7157,E2 231.6356} C_DIS
LIN {X -107.2293,Y -79.1511,Z 179,A -140.8249,B 5.8331,C 0.3271,E1 5.7133,E2 233.0832} C_DIS
LIN {X -109.9023,Y -75.3951,Z 179,A -142.8219,B 5.8333,C 0.3228,E1 5.7101,E2 235.0813} C_DIS
LIN {X -112.327,Y -71.7329,Z 179,A -144.6662,B 5.8336,C 0.3179,E1 5.7073,E2 236.9194} C_DIS
LIN {X -114.1573,Y -68.7829,Z 179,A -146.1734,B 5.8338,C 0.3145,E1 5.7051,E2 238.4279} C_DIS
LIN {X -115.7453,Y -66.0754,Z 179,A -147.5621,B 5.8339,C 0.3116,E1 5.7031,E2 239.8208} C_DIS
LIN {X -117.3148,Y -63.2471,Z 179,A -149.0533,B 5.834,C 0.3092,E1 5.7011,E2 241.3236} C_DIS
LIN {X -118.8163,Y -60.3746,Z 179,A -150.4122,B 5.8342,C 0.3053,E1 5.6994,E2 242.6776} C_DIS
LIN {X -120.2528,Y -57.46,Z 179,A -151.8465,B 5.8344,C 0.3022,E1 5.6976,E2 244.1157} C_DIS
LIN {X -121.6345,Y -54.4742,Z 179,A -153.2885,B 5.8346,C 0.2988,E1 5.696,E2 245.5603} C_DIS
LIN {X -123.1306,Y -51.004,Z 179,A -155.019,B 5.8347,C 0.2956,E1 5.6941,E2 247.3028} C_DIS
LIN {X -124.7511,Y -46.8999,Z 179,A -156.9847,B 5.835,C 0.2912,E1 5.6921,E2 249.2758} C_DIS
LIN {X -126.1951,Y -42.8703,Z 179,A -158.9517,B 5.8351,C 0.2875,E1 5.6903,E2 251.2572} C_DIS
LIN {X -127.3868,Y -39.18,Z 179,A -160.5782,B 5.8354,C 0.2826,E1 5.6889,E2 252.8777} C_DIS
LIN {X -128.4456,Y -35.5569,Z 179,A -162.1456,B 5.8356,C 0.2777,E1 5.6877,E2 254.4375} C_DIS
LIN {X -129.4323,Y -31.7814,Z 179,A -163.7684,B 5.8359,C 0.2726,E1 5.6866,E2 256.0525} C_DIS
LIN {X -130.1881,Y -28.5251,Z 179,A -165.4415,B 5.8359,C 0.2708,E1 5.6855,E2 257.7532} C_DIS
LIN {X -130.9302,Y -24.8953,Z 179,A -166.9706,B 5.8362,C 0.2658,E1 5.6847,E2 259.2736} C_DIS
LIN {X -131.5853,Y -21.1755,Z 179,A -168.6213,B 5.8364,C 0.2615,E1 5.6839,E2 260.9265} C_DIS
LIN {X -132.0642,Y -17.9426,Z 179,A -170.0045,B 5.8365,C 0.2573,E1 5.6834,E2 262.306} C_DIS
LIN {X -132.465,Y -14.6878,Z 179,A -171.5048,B 5.8367,C 0.2542,E1 5.6829,E2 263.8162} C_DIS
LIN {X -132.8277,Y -10.9274,Z 179,A -173.2978,B 5.8368,C 0.2511,E1 5.6825,E2 265.6283} C_DIS
LIN {X -133.1155,Y -6.5439,Z 179,A -175.1831,B 5.837,C 0.2457,E1 5.6821,E2 267.5119} C_DIS
LIN {X -133.259,Y -2.1413,Z 179,A -177.0929,B 5.8373,C 0.2404,E1 5.6821,E2 269.4221} C_DIS
LIN {X -133.259,Y 2.1456,Z 179,A -179.0408,B 5.8374,C 0.2361,E1 5.6821,E2 271.3812} C_DIS
LIN {X -133.1665,Y 5.4116,Z 179,A 179.4987,B 5.8376,C 0.2326,E1 5.6821,E2 272.8473} C_DIS
LIN {X -132.9155,Y 9.7988,Z 179,A 177.6632,B 5.8378,C 0.2268,E1 5.6825,E2 274.6749} C_DIS
LIN {X -132.5681,Y 13.7289,Z 179,A 175.8035,B 5.8379,C 0.2234,E1 5.683,E2 276.5528} C_DIS
LIN {X -132.1316,Y 17.4283,Z 179,A 174.281,B 5.8381,C 0.2182,E1 5.6835,E2 278.0645} C_DIS
LIN {X -131.587,Y 21.1652,Z 179,A 172.6289,B 5.8383,C 0.2139,E1 5.6842,E2 279.7187} C_DIS
LIN {X -131.0277,Y 24.3853,Z 179,A 171.0084,B 5.8383,C 0.2119,E1 5.6851,E2 281.3638} C_DIS
LIN {X -130.1495,Y 28.7043,Z 179,A 169.1107,B 5.8386,C 0.2066,E1 5.6862,E2 283.2603} C_DIS
LIN {X -129.153,Y 32.8933,Z 179,A 167.2599,B 5.8387,C 0.2014,E1 5.6874,E2 285.1094} C_DIS
LIN {X -128.1426,Y 36.6403,Z 179,A 165.3809,B 5.8388,C 0.1988,E1 5.6888,E2 287.0121} C_DIS
LIN {X -126.8987,Y 40.7331,Z 179,A 163.6711,B 5.839,C 0.1926,E1 5.6902,E2 288.7048} C_DIS
LIN {X -125.6627,Y 44.4065,Z 179,A 162.0362,B 5.8392,C 0.1878,E1 5.6917,E2 290.3347} C_DIS
LIN {X -123.9395,Y 49.0104,Z 179,A 159.8637,B 5.8393,C 0.1827,E1 5.6939,E2 292.5124} C_DIS
LIN {X -122.7945,Y 51.8088,Z 179,A 158.3833,B 5.8394,C 0.1809,E1 5.6955,E2 294.0129} C_DIS
LIN {X -121.1724,Y 55.4966,Z 179,A 156.7682,B 5.8396,C 0.1753,E1 5.6973,E2 295.6127} C_DIS
LIN {X -119.9485,Y 58.0971,Z 179,A 155.4027,B 5.8396,C 0.1733,E1 5.699,E2 296.9925} C_DIS
LIN {X -118.2984,Y 61.3865,Z 179,A 153.9071,B 5.8398,C 0.1685,E1 5.7009,E2 298.4764} C_DIS
LIN {X -116.798,Y 64.1977,Z 179,A 152.4646,B 5.8398,C 0.1657,E1 5.7028,E2 299.9264} C_DIS
LIN {X -114.897,Y 67.5398,Z 179,A 150.6768,B 5.8399,C 0.1629,E1 5.7053,E2 301.7287} C_DIS
LIN {X -112.6118,Y 71.285,Z 179,A 148.8616,B 5.8401,C 0.1577,E1 5.708,E2 303.5338} C_DIS
LIN {X -110.8347,Y 74.0176,Z 179,A 147.3381,B 5.8401,C 0.1555,E1 5.7103,E2 305.0705} C_DIS
LIN {X -108.3102,Y 77.665,Z 179,A 145.388,B 5.8402,C 0.1515,E1 5.7135,E2 307.024} C_DIS
LIN {X -106.0671,Y 80.702,Z 179,A 143.8675,B 5.8404,C 0.1468,E1 5.716,E2 308.5309} C_DIS
LIN {X -104.0552,Y 83.2801,Z 179,A 142.2726,B 5.8404,C 0.1454,E1 5.7188,E2 310.1469} C_DIS
LIN {X -101.299,Y 86.6117,Z 179,A 140.3703,B 5.8404,C 0.1418,E1 5.7222,E2 312.0527} C_DIS
LIN {X -98.3701,Y 89.9244,Z 179,A 138.45,B 5.8406,C 0.138,E1 5.7258,E2 313.9736} C_DIS
LIN {X -95.3912,Y 93.0783,Z 179,A 136.543,B 5.8406,C 0.1346,E1 5.7295,E2 315.884} C_DIS
LIN {X -92.4941,Y 95.9575,Z 179,A 134.7552,B 5.8407,C 0.1314,E1 5.7331,E2 317.674} C_DIS
LIN {X -89.501,Y 98.7548,Z 179,A 132.9814,B 5.8407,C 0.1281,E1 5.7367,E2 319.4479} C_DIS
LIN {X -86.4325,Y 101.4513,Z 179,A 131.302,B 5.8409,C 0.1241,E1 5.7402,E2 321.1167} C_DIS
LIN {X -83.4809,Y 103.8938,Z 179,A 129.5231,B 5.8409,C 0.1225,E1 5.7441,E2 322.9097} C_DIS
LIN {X -79.9453,Y 106.6389,Z 179,A 127.629,B 5.8409,C 0.1188,E1 5.7483,E2 324.7988} C_DIS
LIN {X -77.5624,Y 108.3836,Z 179,A 126.2834,B 5.841,C 0.1175,E1 5.7514,E2 326.1523} C_DIS
LIN {X -74.0072,Y 110.8416,Z 179,A 124.5005,B 5.841,C 0.1138,E1 5.7555,E2 327.9249} C_DIS
LIN {X -71.2822,Y 112.6135,Z 179,A 122.9865,B 5.8411,C 0.1129,E1 5.7591,E2 329.4515} C_DIS
LIN {X -67.5463,Y 114.8931,Z 179,A 121.1782,B 5.8411,C 0.1094,E1 5.7634,E2 331.2497} C_DIS
LIN {X -64.7238,Y 116.5066,Z 179,A 119.7655,B 5.8412,C 0.1076,E1 5.7668,E2 332.6631} C_DIS
LIN {X -61.8214,Y 118.07,Z 179,A 118.3252,B 5.8412,C 0.106,E1 5.7704,E2 334.105} C_DIS
LIN {X -58.9092,Y 119.5496,Z 179,A 116.9068,B 5.8412,C 0.1044,E1 5.7739,E2 335.524} C_DIS
LIN {X -55.9613,Y 120.9576,Z 179,A 115.4878,B 5.8412,C 0.1028,E1 5.7775,E2 336.9437} C_DIS
LIN {X -52.9677,Y 122.2981,Z 179,A 113.9783,B 5.8413,C 0.1023,E1 5.7814,E2 338.4639} C_DIS
LIN {X -48.9531,Y 123.9618,Z 179,A 112.021,B 5.8413,C 0.1013,E1 5.7865,E2 340.4304} C_DIS
LIN {X -44.886,Y 125.4902,Z 179,A 110.2438,B 5.8413,C 0.0985,E1 5.7911,E2 342.1957} C_DIS
LIN {X -40.7423,Y 126.8958,Z 179,A 108.3996,B 5.8413,C 0.0965,E1 5.796,E2 344.0342} C_DIS
LIN {X -37.1153,Y 128.004,Z 179,A 106.6948,B 5.8414,C 0.096,E1 5.8005,E2 345.7467} C_DIS
LIN {X -32.8768,Y 129.1572,Z 179,A 104.7743,B 5.8414,C 0.0951,E1 5.8057,E2 347.6698} C_DIS
LIN {X -29.2023,Y 130.0382,Z 179,A 103.2264,B 5.8414,C 0.0932,E1 5.8099,E2 349.2078} C_DIS
LIN {X -26.4866,Y 130.6175,Z 179,A 102.0245,B 5.8414,C 0.0926,E1 5.8132,E2 350.4099} C_DIS
LIN {X -23.2784,Y 131.2274,Z 179,A 100.5654,B 5.8414,C 0.0926,E1 5.8172,E2 351.8747} C_DIS
LIN {X -20.1352,Y 131.7465,Z 179,A 99.1535,B 5.8414,C 0.0926,E1 5.8211,E2 353.2908} C_DIS
LIN {X -16.3167,Y 132.2746,Z 179,A 97.5592,B 5.8414,C 0.0912,E1 5.8255,E2 354.8769} C_DIS
LIN {X -13.0515,Y 132.6359,Z 179,A 96.0607,B 5.8414,C 0.0919,E1 5.8297,E2 356.3847} C_DIS
LIN {X -8.6712,Y 132.9946,Z 179,A 94.1522,B 5.8414,C 0.0917,E1 5.8351,E2 358.2946} C_DIS
LIN {X -4.3958,Y 133.2055,Z 179,A 92.267,B 5.8414,C 0.0921,E1 5.8403,E2 360.1841} C_DIS
LIN {X 0.0164,Y 133.2782,Z 179,A 90.3838,B 5.8414,C 0.092,E1 5.8456,E2 362.0649} C_DIS
LIN {X 4.4085,Y 133.2051,Z 179,A 88.5011,B 5.8414,C 0.0921,E1 5.8508,E2 363.9461} C_DIS
LIN {X 8.6824,Y 132.9939,Z 179,A 86.6732,B 5.8414,C 0.0923,E1 5.8559,E2 365.7719} C_DIS
LIN {X 12.5695,Y 132.6821,Z 179,A 85.1286,B 5.8414,C 0.0912,E1 5.8602,E2 367.3004} C_DIS
LIN {X 15.8186,Y 132.334,Z 179,A 83.7329,B 5.8414,C 0.0915,E1 5.864,E2 368.6945} C_DIS
LIN {X 19.0569,Y 131.9067,Z 179,A 82.2846,B 5.8414,C 0.0927,E1 5.8681,E2 370.1475} C_DIS
LIN {X 22.7853,Y 131.3157,Z 179,A 80.5765,B 5.8414,C 0.0946,E1 5.8728,E2 371.8652} C_DIS
LIN {X 26.7028,Y 130.5735,Z 179,A 78.9628,B 5.8414,C 0.0943,E1 5.8772,E2 373.4665} C_DIS
LIN {X 30.3047,Y 129.7864,Z 179,A 77.4576,B 5.8414,C 0.0943,E1 5.8813,E2 374.962} C_DIS
LIN {X 33.1846,Y 129.0791,Z 179,A 76.1052,B 5.8414,C 0.0962,E1 5.885,E2 376.3231} C_DIS
LIN {X 36.7408,Y 128.1136,Z 179,A 74.4702,B 5.8414,C 0.0981,E1 5.8894,E2 377.9638} C_DIS
LIN {X 40.7494,Y 126.8935,Z 179,A 72.7458,B 5.8414,C 0.0987,E1 5.8939,E2 379.6787} C_DIS
LIN {X 44.4397,Y 125.6511,Z 179,A 70.9097,B 5.8413,C 0.1025,E1 5.8988,E2 381.5337} C_DIS
LIN {X 49.0242,Y 123.9341,Z 179,A 69.0572,B 5.8413,C 0.1013,E1 5.9036,E2 383.3562} C_DIS
LIN {X 51.7673,Y 122.8118,Z 179,A 67.6466,B 5.8413,C 0.1046,E1 5.9073,E2 384.7828} C_DIS
LIN {X 55.4982,Y 121.1717,Z 179,A 66.0704,B 5.8413,C 0.1043,E1 5.9112,E2 386.338} C_DIS
LIN {X 58.4515,Y 119.7754,Z 179,A 64.7712,B 5.8413,C 0.1047,E1 5.9145,E2 387.6248} C_DIS
LIN {X 60.9393,Y 118.5288,Z 179,A 63.4267,B 5.8412,C 0.1082,E1 5.9179,E2 388.9867} C_DIS
LIN {X 64.2757,Y 116.7548,Z 179,A 61.8941,B 5.8412,C 0.1092,E1 5.9216,E2 390.5084} C_DIS
LIN {X 67.1173,Y 115.145,Z 179,A 60.4973,B 5.8412,C 0.1111,E1 5.925,E2 391.9043} C_DIS
LIN {X 69.4856,Y 113.731,Z 179,A 59.2342,B 5.8411,C 0.114,E1 5.928,E2 393.1766} C_DIS
LIN {X 72.6777,Y 111.7179,Z 179,A 57.7299,B 5.8411,C 0.1149,E1 5.9315,E2 394.667} C_DIS
LIN {X 75.8102,Y 109.617,Z 179,A 56.0038,B 5.841,C 0.119,E1 5.9355,E2 396.4056} C_DIS
LIN {X 79.394,Y 107.0494,Z 179,A 54.2683,B 5.841,C 0.1199,E1 5.9394,E2 398.1224} C_DIS
LIN {X 82.4413,Y 104.7205,Z 179,A 52.6012,B 5.841,C 0.1231,E1 5.9431,E2 399.7918} C_DIS
LIN {X 85.6148,Y 102.1423,Z 179,A 50.913,B 5.8409,C 0.1253,E1 5.9467,E2 401.4719} C_DIS
LIN {X 88.3015,Y 99.8288,Z 179,A 49.3166,B 5.8408,C 0.1292,E1 5.9501,E2 403.0773} C_DIS
LIN {X 91.4986,Y 96.9069,Z 179,A 47.4849,B 5.8407,C 0.1324,E1 5.9539,E2 404.9057} C_DIS
LIN {X 94.6369,Y 93.8446,Z 179,A 45.6407,B 5.8407,C 0.1356,E1 5.9575,E2 406.7454} C_DIS
LIN {X 97.6486,Y 90.7067,Z 179,A 43.7874,B 5.8405,C 0.1393,E1 5.9611,E2 408.5972} C_DIS
LIN {X 100.3829,Y 87.671,Z 179,A 42.075,B 5.8405,C 0.1424,E1 5.9642,E2 410.3049} C_DIS
LIN {X 103.0267,Y 84.5488,Z 179,A 40.3882,B 5.8404,C 0.1452,E1 5.9672,E2 411.9836} C_DIS
LIN {X 105.566,Y 81.3565,Z 179,A 38.6562,B 5.8404,C 0.1488,E1 5.9702,E2 413.7137} C_DIS
LIN {X 107.7258,Y 78.4741,Z 179,A 37.1014,B 5.8402,C 0.1525,E1 5.9728,E2 415.2698} C_DIS
LIN {X 109.9023,Y 75.395,Z 179,A 35.5341,B 5.8402,C 0.1555,E1 5.9753,E2 416.8313} C_DIS
LIN {X 112.3251,Y 71.7359,Z 179,A 33.7656,B 5.8401,C 0.1583,E1 5.978,E2 418.5863} C_DIS
LIN {X 114.3132,Y 68.524,Z 179,A 32.2559,B 5.84,C 0.1605,E1 5.9801,E2 420.0831} C_DIS
LIN {X 115.7036,Y 66.1486,Z 179,A 31.0213,B 5.8399,C 0.1642,E1 5.9819,E2 421.3244} C_DIS
LIN {X 117.29,Y 63.2934,Z 179,A 29.5748,B 5.8398,C 0.1683,E1 5.9838,E2 422.7765} C_DIS
LIN {X 118.8192,Y 60.3689,Z 179,A 28.2566,B 5.8398,C 0.1704,E1 5.9855,E2 424.0833} C_DIS
LIN {X 120.2621,Y 57.4406,Z 179,A 26.8845,B 5.8396,C 0.1735,E1 5.9872,E2 425.4523} C_DIS
LIN {X 121.6338,Y 54.476,Z 179,A 25.4944,B 5.8396,C 0.177,E1 5.9888,E2 426.8415} C_DIS
LIN {X 123.1714,Y 50.9062,Z 179,A 23.8044,B 5.8394,C 0.1816,E1 5.9906,E2 428.5347} C_DIS
LIN {X 124.7613,Y 46.8727,Z 179,A 21.9748,B 5.8392,C 0.1861,E1 5.9924,E2 430.3612} C_DIS
LIN {X 126.1925,Y 42.8781,Z 179,A 20.1238,B 5.8391,C 0.1914,E1 5.9941,E2 432.2165} C_DIS
LIN {X 127.3883,Y 39.1751,Z 179,A 18.5522,B 5.839,C 0.1944,E1 5.9955,E2 433.7768} C_DIS
LIN {X 128.4483,Y 35.5474,Z 179,A 17.0553,B 5.8389,C 0.1969,E1 5.9966,E2 435.2594} C_DIS
LIN {X 129.2815,Y 32.3872,Z 179,A 15.6032,B 5.8387,C 0.2015,E1 5.9976,E2 436.718} C_DIS
LIN {X 130.2186,Y 28.3843,Z 179,A 13.8948,B 5.8386,C 0.2055,E1 5.9987,E2 438.4205} C_DIS
LIN {X 130.9304,Y 24.8944,Z 179,A 12.4638,B 5.8385,C 0.2082,E1 5.9994,E2 439.8404} C_DIS
LIN {X 131.5851,Y 21.1764,Z 179,A 10.8928,B 5.8384,C 0.212,E1 6.0002,E2 441.4062} C_DIS
LIN {X 132.0665,Y 17.9253,Z 179,A 9.4876,B 5.8382,C 0.2159,E1 6.0007,E2 442.8115} C_DIS
LIN {X 132.4653,Y 14.685,Z 179,A 8.1339,B 5.8381,C 0.2191,E1 6.0011,E2 444.1601} C_DIS
LIN {X 132.7849,Y 11.4345,Z 179,A 6.7546,B 5.838,C 0.2227,E1 6.0015,E2 445.5374} C_DIS
LIN {X 133.0251,Y 8.1766,Z 179,A 5.3882,B 5.8378,C 0.2261,E1 6.0018,E2 446.9001} C_DIS
LIN {X 133.2059,Y 4.3808,Z 179,A 3.6428,B 5.8376,C 0.2325,E1 6.002,E2 448.6605} C_DIS
LIN {X 133.2794,Y -0.0041,Z 179,A 1.7872,B 5.8374,C 0.2374,E1 6.002,E2 450.514} C_DIS
LIN {X 133.2056,Y -4.3911,Z 179,A -0.0208,B 5.8372,C 0.2416,E1 6.0019,E2 452.3139} C_DIS
LIN {X 132.9931,Y -8.6951,Z 179,A -1.8226,B 5.837,C 0.2461,E1 6.0016,E2 454.1109} C_DIS
LIN {X 132.6829,Y -12.5622,Z 179,A -3.324,B 5.837,C 0.2483,E1 6.0012,E2 455.5933} C_DIS
LIN {X 132.3351,Y -15.809,Z 179,A -4.6895,B 5.8368,C 0.2516,E1 6.0008,E2 456.9553} C_DIS
LIN {X 131.9082,Y -19.0465,Z 179,A -6.1058,B 5.8366,C 0.2558,E1 6.0002,E2 458.3743} C_DIS
LIN {X 131.4023,Y -22.2718,Z 179,A -7.504,B 5.8364,C 0.2597,E1 5.9996,E2 459.7731} C_DIS
LIN {X 130.7163,Y -26.0015,Z 179,A -9.0287,B 5.8364,C 0.2627,E1 5.9988,E2 461.2863} C_DIS
LIN {X 130.1495,Y -28.7039,Z 179,A -10.174,B 5.8362,C 0.2654,E1 5.9982,E2 462.4275} C_DIS
LIN {X 129.2832,Y -32.3803,Z 179,A -11.7377,B 5.836,C 0.269,E1 5.9971,E2 463.9852} C_DIS
LIN {X 128.6646,Y -34.7569,Z 179,A -12.861,B 5.8358,C 0.2729,E1 5.9963,E2 465.1177} C_DIS
LIN {X 127.3906,Y -39.1677,Z 179,A -14.7278,B 5.8357,C 0.2767,E1 5.9948,E2 466.9731} C_DIS
LIN {X 126.1879,Y -42.8916,Z 179,A -16.3631,B 5.8355,C 0.2806,E1 5.9934,E2 468.6041} C_DIS
LIN {X 124.7469,Y -46.9113,Z 179,A -18.2286,B 5.8352,C 0.286,E1 5.9916,E2 470.4749} C_DIS
LIN {X 123.3246,Y -50.5375,Z 179,A -19.884,B 5.835,C 0.2902,E1 5.9899,E2 472.1295} C_DIS
LIN {X 121.8432,Y -54.0077,Z 179,A -21.3775,B 5.8349,C 0.2925,E1 5.9883,E2 473.6086} C_DIS
LIN {X 120.4833,Y -56.9776,Z 179,A -22.7485,B 5.8347,C 0.2957,E1 5.9866,E2 474.9768} C_DIS
LIN {X 119.0516,Y -59.9124,Z 179,A -24.119,B 5.8346,C 0.2988,E1 5.985,E2 476.3444} C_DIS
LIN {X 117.3126,Y -63.2512,Z 179,A -25.7755,B 5.8343,C 0.3036,E1 5.9828,E2 478.0072} C_DIS
LIN {X 115.1458,Y -67.1158,Z 179,A -27.579,B 5.8342,C 0.3068,E1 5.9803,E2 479.7999} C_DIS
LIN {X 113.7298,Y -69.4876,Z 179,A -28.8315,B 5.8339,C 0.3108,E1 5.9785,E2 481.0615} C_DIS
LIN {X 111.7172,Y -72.6789,Z 179,A -30.3252,B 5.8339,C 0.3128,E1 5.9763,E2 482.5408} C_DIS
LIN {X 109.6137,Y -75.815,Z 179,A -32.041,B 5.8336,C 0.3181,E1 5.9735,E2 484.2695} C_DIS
LIN {X 107.0458,Y -79.399,Z 179,A -33.7654,B 5.8335,C 0.32,E1 5.9707,E2 485.9744} C_DIS
LIN {X 104.7196,Y -82.4424,Z 179,A -35.4243,B 5.8332,C 0.324,E1 5.9679,E2 487.6363} C_DIS
LIN {X 102.1453,Y -85.6112,Z 179,A -37.1084,B 5.8331,C 0.3269,E1 5.9649,E2 489.3132} C_DIS
LIN {X 99.8342,Y -88.2953,Z 179,A -38.6937,B 5.8328,C 0.3312,E1 5.962,E2 490.9076} C_DIS
LIN {X 96.9091,Y -91.4963,Z 179,A -40.5249,B 5.8326,C 0.3348,E1 5.9585,E2 492.7364} C_DIS
LIN {X 93.8435,Y -94.638,Z 179,A -42.37,B 5.8324,C 0.3381,E1 5.9549,E2 494.578} C_DIS
LIN {X 90.6997,Y -97.6551,Z 179,A -44.227,B 5.8322,C 0.3417,E1 5.9511,E2 496.4346} C_DIS
LIN {X 87.6663,Y -100.387,Z 179,A -45.9385,B 5.8321,C 0.3445,E1 5.9476,E2 498.1422} C_DIS
LIN {X 84.5505,Y -103.0253,Z 179,A -47.6282,B 5.8319,C 0.3469,E1 5.9439,E2 499.8254} C_DIS
LIN {X 81.3556,Y -105.5667,Z 179,A -49.3649,B 5.8317,C 0.3498,E1 5.9401,E2 501.5613} C_DIS
LIN {X 78.4795,Y -107.7219,Z 179,A -50.9263,B 5.8316,C 0.3528,E1 5.9366,E2 503.126} C_DIS
LIN {X 75.3978,Y -109.9004,Z 179,A -52.5028,B 5.8314,C 0.355,E1 5.933,E2 504.6981} C_DIS
LIN {X 71.7359,Y -112.325,Z 179,A -54.2834,B 5.8314,C 0.3565,E1 5.9289,E2 506.4669} C_DIS
LIN {X 68.5265,Y -114.3117,Z 179,A -55.8046,B 5.8313,C 0.3577,E1 5.9253,E2 507.9768} C_DIS
LIN {X 66.1987,Y -115.675,Z 179,A -56.9705,B 5.8312,C 0.3595,E1 5.9225,E2 509.1443} C_DIS
LIN {X 63.2487,Y -117.314,Z 179,A -58.523,B 5.8309,C 0.3631,E1 5.9186,E2 510.7107} C_DIS
LIN {X 60.3615,Y -118.8229,Z 179,A -59.8436,B 5.8309,C 0.3639,E1 5.9154,E2 512.0224} C_DIS
LIN {X 57.4338,Y -120.2653,Z 179,A -61.2294,B 5.8308,C 0.3656,E1 5.9119,E2 513.407} C_DIS
LIN {X 54.471,Y -121.636,Z 179,A -62.6165,B 5.8307,C 0.3672,E1 5.9084,E2 514.7932} C_DIS
LIN {X 50.9824,Y -123.1396,Z 179,A -64.2933,B 5.8305,C 0.3698,E1 5.904,E2 516.4767} C_DIS
LIN {X 47.2438,Y -124.6223,Z 179,A -66.1214,B 5.8303,C 0.3731,E1 5.8992,E2 518.3183} C_DIS
LIN {X 43.3685,Y -126.0226,Z 179,A -67.6874,B 5.8303,C 0.3722,E1 5.8952,E2 519.86} C_DIS
LIN {X 40.2516,Y -127.0525,Z 179,A -69.0995,B 5.8303,C 0.3736,E1 5.8914,E2 521.2732} C_DIS
LIN {X 37.1115,Y -128.0051,Z 179,A -70.5599,B 5.8302,C 0.3756,E1 5.8875,E2 522.7407} C_DIS
LIN {X 32.8714,Y -129.1586,Z 179,A -72.4528,B 5.83,C 0.3772,E1 5.8824,E2 524.6353} C_DIS
LIN {X 29.2001,Y -130.0387,Z 179,A -73.981,B 5.83,C 0.3772,E1 5.8782,E2 526.1528} C_DIS
LIN {X 26.5034,Y -130.6141,Z 179,A -75.167,B 5.83,C 0.378,E1 5.875,E2 527.3396} C_DIS
LIN {X 23.2688,Y -131.2292,Z 179,A -76.6184,B 5.83,C 0.3794,E1 5.871,E2 528.7963} C_DIS
LIN {X 20.0486,Y -131.7599,Z 179,A -78.0406,B 5.8298,C 0.3804,E1 5.8671,E2 530.2218} C_DIS
LIN {X 16.7269,Y -132.2236,Z 179,A -79.4982,B 5.8298,C 0.3814,E1 5.863,E2 531.6822} C_DIS
LIN {X 13.0669,Y -132.6344,Z 179,A -81.0852,B 5.8298,C 0.3821,E1 5.8586,E2 533.2704} C_DIS
LIN {X 8.659,Y -132.9954,Z 179,A -82.9891,B 5.8297,C 0.3827,E1 5.8533,E2 535.1757} C_DIS
LIN {X 4.3978,Y -133.2054,Z 179,A -84.8664,B 5.8297,C 0.3837,E1 5.848,E2 537.0593} C_DIS
LIN {X 0.9647,Y -133.2696,Z 179,A -85.7807,B 5.8301,C 0.3768,E1 5.8457,E2 537.904} C_DIS
Enddeposition()
LIN {X 0.9647,Y -133.2696,Z 179,A -85.7807,B 5.8301,C 0.3768,E1 5.8457,E2 537.904} C_DIS
Startdeposition()
$VEL.CP = VEL_PRINT
LIN {X 1.8565,Y -134.1672,Z 179,A -85.0305,B 5.8301,C 0.3752,E1 5.8477,E2 537.1393} C_DIS
LIN {X 6.3876,Y -134.0278,Z 179,A -83.1801,B 5.8301,C 0.3759,E1 5.8528,E2 535.2988} C_DIS
LIN {X 9.1575,Y -133.868,Z 179,A -81.8491,B 5.8301,C 0.3736,E1 5.8566,E2 533.9486} C_DIS
LIN {X 13.7139,Y -133.4783,Z 179,A -79.974,B 5.8301,C 0.3738,E1 5.8618,E2 532.0824} C_DIS
LIN {X 17.3714,Y -133.0502,Z 179,A -78.5349,B 5.8301,C 0.3749,E1 5.8657,E2 530.6593} C_DIS
LIN {X 20.5734,Y -132.5927,Z 179,A -77.1731,B 5.8301,C 0.3744,E1 5.8695,E2 529.2992} C_DIS
LIN {X 23.5166,Y -132.1025,Z 179,A -75.7208,B 5.8303,C 0.3712,E1 5.8735,E2 527.8235} C_DIS
LIN {X 27.8799,Y -131.2516,Z 179,A -74.0734,B 5.8302,C 0.3733,E1 5.878,E2 526.2068} C_DIS
LIN {X 31.0258,Y -130.5437,Z 179,A -72.7092,B 5.8302,C 0.3724,E1 5.8817,E2 524.8433} C_DIS
LIN {X 34.5085,Y -129.6658,Z 179,A -71.0794,B 5.8304,C 0.3698,E1 5.8861,E2 523.2003} C_DIS
LIN {X 37.8705,Y -128.7241,Z 179,A -69.6001,B 5.8304,C 0.3687,E1 5.8901,E2 521.7215} C_DIS
LIN {X 41.3518,Y -127.6494,Z 179,A -68.2036,B 5.8304,C 0.3694,E1 5.8938,E2 520.3441} C_DIS
LIN {X 45.6065,Y -126.1907,Z 179,A -66.169,B 5.8307,C 0.3657,E1 5.8992,E2 518.2938} C_DIS
LIN {X 48.2688,Y -125.197,Z 179,A -64.4998,B 5.8311,C 0.3579,E1 5.9037,E2 516.5656} C_DIS
LIN {X 52.1972,Y -123.6112,Z 179,A -63.023,B 5.831,C 0.3605,E1 5.9074,E2 515.1299} C_DIS
LIN {X 55.5802,Y -122.129,Z 179,A -61.4331,B 5.8311,C 0.3583,E1 5.9114,E2 513.5372} C_DIS
LIN {X 58.8355,Y -120.5932,Z 179,A -60.0346,B 5.8311,C 0.3582,E1 5.9149,E2 512.1552} C_DIS
LIN {X 61.8154,Y -119.0934,Z 179,A -58.6047,B 5.8312,C 0.3561,E1 5.9185,E2 510.7235} C_DIS
LIN {X 65.8652,Y -116.9031,Z 179,A -56.6636,B 5.8314,C 0.3536,E1 5.9232,E2 508.7841} C_DIS
LIN {X 69.7686,Y -114.6169,Z 179,A -54.7552,B 5.8316,C 0.3509,E1 5.9278,E2 506.8771} C_DIS
LIN {X 73.3738,Y -112.343,Z 179,A -53.0531,B 5.8316,C 0.3496,E1 5.9318,E2 505.1884} C_DIS
LIN {X 76.2035,Y -110.4431,Z 179,A -51.51,B 5.8319,C 0.3459,E1 5.9353,E2 503.633} C_DIS
LIN {X 79.7942,Y -107.8777,Z 179,A -49.7273,B 5.8319,C 0.3441,E1 5.9393,E2 501.8617} C_DIS
LIN {X 83.0275,Y -105.4087,Z 179,A -47.9697,B 5.8322,C 0.3406,E1 5.9432,E2 500.1} C_DIS
LIN {X 86.2929,Y -102.7525,Z 179,A -46.2375,B 5.8323,C 0.3381,E1 5.9469,E2 498.3745} C_DIS
LIN {X 89.476,Y -99.9929,Z 179,A -44.4391,B 5.8325,C 0.3346,E1 5.9507,E2 496.5746} C_DIS
LIN {X 93.3895,Y -96.348,Z 179,A -42.2005,B 5.8327,C 0.3306,E1 5.9553,E2 494.3397} C_DIS
LIN {X 96.4172,Y -93.318,Z 179,A -40.436,B 5.8329,C 0.3278,E1 5.9587,E2 492.5817} C_DIS
LIN {X 99.1986,Y -90.3562,Z 179,A -38.702,B 5.8331,C 0.324,E1 5.962,E2 490.8463} C_DIS
LIN {X 101.9842,Y -87.2003,Z 179,A -36.8802,B 5.8334,C 0.3197,E1 5.9653,E2 489.0199} C_DIS
LIN {X 104.7681,Y -83.835,Z 179,A -35.0544,B 5.8336,C 0.316,E1 5.9685,E2 487.1973} C_DIS
LIN {X 107.2528,Y -80.6315,Z 179,A -33.4771,B 5.8336,C 0.3143,E1 5.9712,E2 485.6379} C_DIS
LIN {X 109.565,Y -77.4601,Z 179,A -31.742,B 5.8339,C 0.3095,E1 5.974,E2 483.8939} C_DIS
LIN {X 111.8574,Y -74.1121,Z 179,A -30.0108,B 5.8341,C 0.3053,E1 5.9767,E2 482.1612} C_DIS
LIN {X 114.1714,Y -70.4952,Z 179,A -28.2188,B 5.8343,C 0.3014,E1 5.9794,E2 480.3728} C_DIS
LIN {X 116.5029,Y -66.5704,Z 179,A -26.3534,B 5.8345,C 0.2978,E1 5.982,E2 478.5162} C_DIS
LIN {X 119.2364,Y -61.5405,Z 179,A -24.0131,B 5.8347,C 0.2932,E1 5.985,E2 476.1869} C_DIS
LIN {X 120.985,Y -58.0229,Z 179,A -22.4139,B 5.8349,C 0.29,E1 5.987,E2 474.5958} C_DIS
LIN {X 122.2415,Y -55.3298,Z 179,A -21.2623,B 5.8349,C 0.2885,E1 5.9883,E2 473.458} C_DIS
LIN {X 123.6421,Y -52.1234,Z 179,A -19.6159,B 5.8353,C 0.2822,E1 5.9901,E2 471.791} C_DIS
LIN {X 124.7741,Y -49.3566,Z 179,A -18.3839,B 5.8354,C 0.2795,E1 5.9914,E2 470.5636} C_DIS
LIN {X 126.1909,Y -45.6057,Z 179,A -16.8206,B 5.8355,C 0.2772,E1 5.9929,E2 469.0173} C_DIS
LIN {X 127.2264,Y -42.6325,Z 179,A -15.3047,B 5.8358,C 0.2708,E1 5.9943,E2 467.4787} C_DIS
LIN {X 128.5078,Y -38.6038,Z 179,A -13.7285,B 5.8358,C 0.2695,E1 5.9956,E2 465.9297} C_DIS
LIN {X 130.2603,Y -32.2015,Z 179,A -10.8364,B 5.8363,C 0.2607,E1 5.9977,E2 463.0281} C_DIS
LIN {X 131.0362,Y -28.8778,Z 179,A -9.4221,B 5.8364,C 0.2573,E1 5.9985,E2 461.6179} C_DIS
LIN {X 131.9317,Y -24.4672,Z 179,A -7.6732,B 5.8365,C 0.2546,E1 5.9994,E2 459.889} C_DIS
LIN {X 132.512,Y -21.0947,Z 179,A -6.1032,B 5.8368,C 0.2488,E1 6.0002,E2 458.3041} C_DIS
LIN {X 133.068,Y -17.2352,Z 179,A -4.5356,B 5.8369,C 0.2456,E1 6.0007,E2 456.7473} C_DIS
LIN {X 133.5167,Y -13.3297,Z 179,A -2.8855,B 5.8371,C 0.2412,E1 6.0012,E2 455.0994} C_DIS
LIN {X 133.8368,Y -9.5848,Z 179,A -1.5191,B 5.8371,C 0.2404,E1 6.0015,E2 453.7613} C_DIS
LIN {X 134.0758,Y -5.2739,Z 179,A 0.4703,B 5.8374,C 0.2329,E1 6.0018,E2 451.7523} C_DIS
LIN {X 134.177,Y -0.9519,Z 179,A 2.2813,B 5.8376,C 0.2281,E1 6.0018,E2 449.9443} C_DIS
LIN {X 134.1408,Y 3.2594,Z 179,A 3.9187,B 5.8377,C 0.2255,E1 6.0018,E2 448.3256} C_DIS
LIN {X 133.9978,Y 6.9845,Z 179,A 5.622,B 5.838,C 0.2192,E1 6.0016,E2 446.6072} C_DIS
LIN {X 133.6888,Y 11.4655,Z 179,A 7.4309,B 5.8381,C 0.2155,E1 6.0012,E2 444.8104} C_DIS
LIN {X 133.3083,Y 15.2772,Z 179,A 9.095,B 5.8383,C 0.2104,E1 6.0007,E2 443.1417} C_DIS
LIN {X 132.7965,Y 19.2157,Z 179,A 10.6511,B 5.8383,C 0.2078,E1 6.0001,E2 441.6016} C_DIS
LIN {X 132.1632,Y 23.1774,Z 179,A 12.3498,B 5.8386,C 0.2032,E1 5.9993,E2 439.9035} C_DIS
LIN {X 131.575,Y 26.3116,Z 179,A 13.6959,B 5.8386,C 0.1997,E1 5.9986,E2 438.5584} C_DIS
LIN {X 130.8016,Y 29.9169,Z 179,A 15.1772,B 5.8388,C 0.1967,E1 5.9977,E2 437.0876} C_DIS
LIN {X 129.8572,Y 33.7905,Z 179,A 16.9756,B 5.839,C 0.1906,E1 5.9965,E2 435.2763} C_DIS
LIN {X 128.8752,Y 37.3546,Z 179,A 18.3569,B 5.839,C 0.1893,E1 5.9955,E2 433.9184} C_DIS
LIN {X 127.8824,Y 40.6223,Z 179,A 20.0308,B 5.8392,C 0.182,E1 5.994,E2 432.217} C_DIS
LIN {X 126.416,Y 44.9815,Z 179,A 22.4047,B 5.8396,C 0.1703,E1 5.9918,E2 429.7911} C_DIS
LIN {X 124.5369,Y 49.9464,Z 179,A 24.2953,B 5.8396,C 0.1702,E1 5.9899,E2 427.946} C_DIS
LIN {X 123.1569,Y 53.2578,Z 179,A 25.4879,B 5.8396,C 0.1714,E1 5.9886,E2 426.7944} C_DIS
LIN {X 121.4843,Y 56.9744,Z 179,A 27.1415,B 5.8396,C 0.1682,E1 5.9867,E2 425.1506} C_DIS
LIN {X 119.7237,Y 60.5832,Z 179,A 28.8481,B 5.8398,C 0.164,E1 5.9846,E2 423.4441} C_DIS
LIN {X 117.9067,Y 64.0515,Z 179,A 30.5631,B 5.8399,C 0.1591,E1 5.9823,E2 421.7231} C_DIS
LIN {X 115.7086,Y 67.9416,Z 179,A 32.3712,B 5.84,C 0.1559,E1 5.9798,E2 419.9263} C_DIS
LIN {X 113.7597,Y 71.1574,Z 179,A 34.0099,B 5.8401,C 0.1515,E1 5.9774,E2 418.283} C_DIS
LIN {X 111.2776,Y 74.9795,Z 179,A 35.9087,B 5.8402,C 0.1476,E1 5.9745,E2 416.3892} C_DIS
LIN {X 108.7548,Y 78.5937,Z 179,A 37.7458,B 5.8403,C 0.1439,E1 5.9715,E2 414.5569} C_DIS
LIN {X 106.0804,Y 82.1674,Z 179,A 39.5846,B 5.8403,C 0.1406,E1 5.9684,E2 412.7256} C_DIS
LIN {X 103.5447,Y 85.3412,Z 179,A 41.2627,B 5.8405,C 0.1376,E1 5.9655,E2 411.0539} C_DIS
LIN {X 100.8786,Y 88.4768,Z 179,A 43.0127,B 5.8405,C 0.1339,E1 5.9623,E2 409.3043} C_DIS
LIN {X 97.9815,Y 91.6747,Z 179,A 44.6179,B 5.8405,C 0.1335,E1 5.9593,E2 407.7275} C_DIS
LIN {X 95.5244,Y 94.2325,Z 179,A 46.3668,B 5.8407,C 0.1269,E1 5.9558,E2 405.9497} C_DIS
LIN {X 92.3411,Y 97.3539,Z 179,A 48.239,B 5.8407,C 0.1236,E1 5.9521,E2 404.081} C_DIS
LIN {X 90.1513,Y 99.3845,Z 179,A 49.5874,B 5.8408,C 0.1201,E1 5.9493,E2 402.7234} C_DIS
LIN {X 86.366,Y 102.6912,Z 179,A 51.4973,B 5.8408,C 0.1195,E1 5.9453,E2 400.8419} C_DIS
LIN {X 83.3099,Y 105.186,Z 179,A 53.2155,B 5.8409,C 0.116,E1 5.9415,E2 399.1195} C_DIS
LIN {X 79.9927,Y 107.7299,Z 179,A 54.9487,B 5.8409,C 0.1136,E1 5.9377,E2 397.3923} C_DIS
LIN {X 76.4658,Y 110.2613,Z 179,A 56.7715,B 5.841,C 0.111,E1 5.9335,E2 395.5731} C_DIS
LIN {X 72.9185,Y 112.6386,Z 179,A 58.6198,B 5.841,C 0.1078,E1 5.9292,E2 393.7217} C_DIS
LIN {X 69.3023,Y 114.8989,Z 179,A 60.3854,B 5.8411,C 0.1058,E1 5.925,E2 391.9628} C_DIS
LIN {X 65.4058,Y 117.1613,Z 179,A 62.3467,B 5.8411,C 0.1025,E1 5.9202,E2 389.9971} C_DIS
LIN {X 61.3298,Y 119.3437,Z 179,A 64.2145,B 5.8411,C 0.1013,E1 5.9156,E2 388.1421} C_DIS
LIN {X 57.9623,Y 121.014,Z 179,A 65.6548,B 5.8411,C 0.1015,E1 5.9121,E2 386.7218} C_DIS
LIN {X 55.5363,Y 122.1491,Z 179,A 66.8755,B 5.8412,C 0.0991,E1 5.909,E2 385.492} C_DIS
LIN {X 52.2243,Y 123.5999,Z 179,A 68.5075,B 5.8412,C 0.0961,E1 5.9047,E2 383.8494} C_DIS
LIN {X 49.3686,Y 124.7694,Z 179,A 69.8672,B 5.8413,C 0.0942,E1 5.9012,E2 382.4849} C_DIS
LIN {X 45.3451,Y 126.2849,Z 179,A 71.6633,B 5.8413,C 0.0928,E1 5.8965,E2 380.6938} C_DIS
LIN {X 41.7111,Y 127.5333,Z 179,A 73.1523,B 5.8413,C 0.0933,E1 5.8926,E2 379.2234} C_DIS
LIN {X 35.9175,Y 129.2828,Z 179,A 76.1174,B 5.8414,C 0.0862,E1 5.8845,E2 376.2129} C_DIS
LIN {X 32.1744,Y 130.2668,Z 179,A 77.557,B 5.8414,C 0.0878,E1 5.8807,E2 374.7996} C_DIS
LIN {X 27.4975,Y 131.3337,Z 179,A 79.4904,B 5.8414,C 0.088,E1 5.8755,E2 372.8806} C_DIS
LIN {X 24.2733,Y 131.9671,Z 179,A 80.8984,B 5.8414,C 0.0871,E1 5.8716,E2 371.4723} C_DIS
LIN {X 20.6351,Y 132.5832,Z 179,A 82.3893,B 5.8414,C 0.0874,E1 5.8675,E2 369.9921} C_DIS
LIN {X 17.1002,Y 133.0857,Z 179,A 83.9911,B 5.8414,C 0.0858,E1 5.8631,E2 368.3816} C_DIS
LIN {X 13.2991,Y 133.5196,Z 179,A 85.6918,B 5.8414,C 0.0845,E1 5.8583,E2 366.6734} C_DIS
LIN {X 8.508,Y 133.9097,Z 179,A 87.6527,B 5.8414,C 0.0851,E1 5.8529,E2 364.7243} C_DIS
LIN {X 4.7002,Y 134.0982,Z 179,A 89.1671,B 5.8414,C 0.0863,E1 5.8487,E2 363.2242} C_DIS
LIN {X 0.9263,Y 134.1765,Z 179,A 90.8518,B 5.8414,C 0.0853,E1 5.844,E2 361.5315} C_DIS
LIN {X -2.8946,Y 134.15,Z 179,A 92.4923,B 5.8414,C 0.0852,E1 5.8394,E2 359.8906} C_DIS
LIN {X -6.0195,Y 134.046,Z 179,A 93.783,B 5.8414,C 0.0858,E1 5.8358,E2 358.606} C_DIS
LIN {X -9.7946,Y 133.8215,Z 179,A 95.4343,B 5.8414,C 0.0856,E1 5.8312,E2 356.951} C_DIS
LIN {X -13.0096,Y 133.5474,Z 179,A 96.9797,B 5.8414,C 0.084,E1 5.8268,E2 355.3861} C_DIS
LIN {X -17.4083,Y 133.0453,Z 179,A 98.6997,B 5.8414,C 0.0866,E1 5.8221,E2 353.6877} C_DIS
LIN {X -21.3717,Y 132.4683,Z 179,A 100.5621,B 5.8414,C 0.0855,E1 5.8169,E2 351.808} C_DIS
LIN {X -25.6348,Y 131.7085,Z 179,A 102.371,B 5.8414,C 0.0869,E1 5.812,E2 350.005} C_DIS
LIN {X -29.5822,Y 130.878,Z 179,A 104.0236,B 5.8414,C 0.0887,E1 5.8075,E2 348.3617} C_DIS
LIN {X -33.0564,Y 130.0436,Z 179,A 105.503,B 5.8414,C 0.0902,E1 5.8035,E2 346.8888} C_DIS
LIN {X -37.0139,Y 128.9749,Z 179,A 107.2223,B 5.8414,C 0.0919,E1 5.7989,E2 345.1745} C_DIS
LIN {X -41.7626,Y 127.5161,Z 179,A 109.5012,B 5.8414,C 0.0919,E1 5.7928,E2 342.8781} C_DIS
LIN {X -50.3472,Y 124.3753,Z 179,A 113.3728,B 5.8413,C 0.096,E1 5.7827,E2 339.0131} C_DIS
LIN {X -54.3016,Y 122.7013,Z 179,A 115.2183,B 5.8413,C 0.0979,E1 5.7779,E2 337.1675} C_DIS
LIN {X -57.4416,Y 121.2627,Z 179,A 116.7185,B 5.8413,C 0.0994,E1 5.7741,E2 335.6653} C_DIS
LIN {X -60.745,Y 119.6414,Z 179,A 118.2933,B 5.8412,C 0.1013,E1 5.7702,E2 334.0912} C_DIS
LIN {X -66.2293,Y 116.6975,Z 179,A 121.0507,B 5.8412,C 0.1039,E1 5.7634,E2 331.324} C_DIS
LIN {X -69.8905,Y 114.5424,Z 179,A 122.732,B 5.8411,C 0.1079,E1 5.7594,E2 329.6601} C_DIS
LIN {X -73.4333,Y 112.3043,Z 179,A 125.1872,B 5.8411,C 0.1036,E1 5.7535,E2 327.126} C_DIS
LIN {X -77.2398,Y 109.7204,Z 179,A 126.6743,B 5.8411,C 0.1118,E1 5.7502,E2 325.6982} C_DIS
LIN {X -80.6587,Y 107.2322,Z 179,A 128.5564,B 5.841,C 0.114,E1 5.746,E2 323.8084} C_DIS
LIN {X -84.2694,Y 104.4184,Z 179,A 130.4956,B 5.8409,C 0.1176,E1 5.7417,E2 321.8726} C_DIS
LIN {X -87.6419,Y 101.6043,Z 179,A 132.4152,B 5.8409,C 0.1206,E1 5.7376,E2 319.9493} C_DIS
LIN {X -90.8549,Y 98.7417,Z 179,A 134.2938,B 5.8408,C 0.1237,E1 5.7337,E2 318.0673} C_DIS
LIN {X -94.1936,Y 95.5626,Z 179,A 136.3206,B 5.8407,C 0.127,E1 5.7297,E2 316.0352} C_DIS
LIN {X -97.3335,Y 92.3628,Z 179,A 138.2945,B 5.8407,C 0.1303,E1 5.7258,E2 314.0558} C_DIS
LIN {X -100.4103,Y 89.0075,Z 179,A 140.2462,B 5.8405,C 0.1344,E1 5.7222,E2 312.1048} C_DIS
LIN {X -103.3825,Y 85.5371,Z 179,A 142.2094,B 5.8405,C 0.1385,E1 5.7187,E2 310.1419} C_DIS
LIN {X -106.2297,Y 81.9748,Z 179,A 144.2265,B 5.8403,C 0.1422,E1 5.7152,E2 308.1181} C_DIS
LIN {X -108.7257,Y 78.6339,Z 179,A 146.0147,B 5.8403,C 0.1462,E1 5.7122,E2 306.3305} C_DIS
LIN {X -111.122,Y 75.2093,Z 179,A 148.3084,B 5.8403,C 0.1454,E1 5.7085,E2 303.9765} C_DIS
LIN {X -113.6145,Y 71.3887,Z 179,A 149.7952,B 5.84,C 0.1546,E1 5.7064,E2 302.5476} C_DIS
LIN {X -115.5162,Y 68.2692,Z 179,A 151.4335,B 5.84,C 0.1577,E1 5.704,E2 300.9012} C_DIS
LIN {X -117.5442,Y 64.7148,Z 179,A 153.1517,B 5.8398,C 0.1623,E1 5.7017,E2 299.1881} C_DIS
LIN {X -119.409,Y 61.2014,Z 179,A 155.0809,B 5.8398,C 0.1644,E1 5.6992,E2 297.2323} C_DIS
LIN {X -121.5542,Y 56.8233,Z 179,A 156.9918,B 5.8396,C 0.1714,E1 5.6969,E2 295.3441} C_DIS
LIN {X -123.1034,Y 53.3814,Z 179,A 158.6916,B 5.8395,C 0.1748,E1 5.6949,E2 293.635} C_DIS
LIN {X -124.4641,Y 50.1268,Z 179,A 160.1041,B 5.8393,C 0.1797,E1 5.6935,E2 292.2353} C_DIS
LIN {X -125.6283,Y 47.1333,Z 179,A 161.7679,B 5.8393,C 0.1806,E1 5.6918,E2 290.5371} C_DIS
LIN {X -127.2233,Y 42.6418,Z 179,A 163.5068,B 5.839,C 0.1889,E1 5.6902,E2 288.836} C_DIS
LIN {X -128.2033,Y 39.599,Z 179,A 165.0375,B 5.839,C 0.191,E1 5.6889,E2 287.2864} C_DIS
LIN {X -129.0846,Y 36.626,Z 179,A 166.4982,B 5.8389,C 0.1934,E1 5.6878,E2 285.8103} C_DIS
LIN {X -130.2247,Y 32.3428,Z 179,A 168.5013,B 5.8387,C 0.1976,E1 5.6864,E2 283.7953} C_DIS
LIN {X -131.0286,Y 28.9126,Z 179,A 169.9902,B 5.8386,C 0.2019,E1 5.6855,E2 282.3096} C_DIS
LIN {X -131.8129,Y 25.089,Z 179,A 171.6384,B 5.8384,C 0.2068,E1 5.6846,E2 280.6651} C_DIS
LIN {X -132.5201,Y 21.0422,Z 179,A 173.4734,B 5.8383,C 0.211,E1 5.6837,E2 278.8217} C_DIS
LIN {X -133.0367,Y 17.4741,Z 179,A 174.9533,B 5.8381,C 0.2159,E1 5.6832,E2 277.3503} C_DIS
LIN {X -133.3996,Y 14.4457,Z 179,A 176.2436,B 5.838,C 0.2197,E1 5.6828,E2 276.0627} C_DIS
LIN {X -133.7096,Y 11.2196,Z 179,A 177.7548,B 5.8379,C 0.2224,E1 5.6824,E2 274.537} C_DIS
LIN {X -133.9917,Y 7.1054,Z 179,A 179.6182,B 5.8377,C 0.2265,E1 5.682,E2 272.6624} C_DIS
LIN {X -134.148,Y 3.0009,Z 179,A -178.5218,B 5.8375,C 0.2305,E1 5.6819,E2 270.7908} C_DIS
LIN {X -134.1736,Y -1.454,Z 179,A -176.5533,B 5.8373,C 0.2353,E1 5.6819,E2 268.8157} C_DIS
LIN {X -134.0631,Y -5.5996,Z 179,A -174.8934,B 5.8371,C 0.2414,E1 5.6821,E2 267.1707} C_DIS
LIN {X -133.8842,Y -8.923,Z 179,A -173.3055,B 5.837,C 0.2439,E1 5.6823,E2 265.5634} C_DIS
LIN {X -133.5643,Y -12.8331,Z 179,A -171.7142,B 5.8368,C 0.2494,E1 5.6827,E2 263.9836} C_DIS
LIN {X -133.1937,Y -16.2378,Z 179,A -170.0636,B 5.8367,C 0.2518,E1 5.6833,E2 262.3109} C_DIS
LIN {X -132.6259,Y -20.3591,Z 179,A -168.3432,B 5.8364,C 0.2573,E1 5.684,E2 260.5986} C_DIS
LIN {X -132.0061,Y -24.0551,Z 179,A -166.6269,B 5.8363,C 0.2607,E1 5.6848,E2 258.8692} C_DIS
LIN {X -131.1394,Y -28.3997,Z 179,A -164.9232,B 5.836,C 0.2677,E1 5.6858,E2 257.19} C_DIS
LIN {X -130.077,Y -32.9246,Z 179,A -162.7016,B 5.8358,C 0.271,E1 5.6872,E2 254.9404} C_DIS
LIN {X -128.9295,Y -37.1689,Z 179,A -160.7884,B 5.8356,C 0.2757,E1 5.6887,E2 253.024} C_DIS
LIN {X -127.9204,Y -40.5035,Z 179,A -159.1921,B 5.8354,C 0.2787,E1 5.69,E2 251.4151} C_DIS
LIN {X -126.58,Y -44.5183,Z 179,A -157.4428,B 5.8352,C 0.2841,E1 5.6916,E2 249.6741} C_DIS
LIN {X -125.5406,Y -47.3675,Z 179,A -156.0611,B 5.8351,C 0.2867,E1 5.6929,E2 248.2824} C_DIS
LIN {X -123.985,Y -51.3023,Z 179,A -154.2038,B 5.8349,C 0.2909,E1 5.6949,E2 246.4198} C_DIS
Enddeposition()
END
